ABB RAPID module: P705.mod

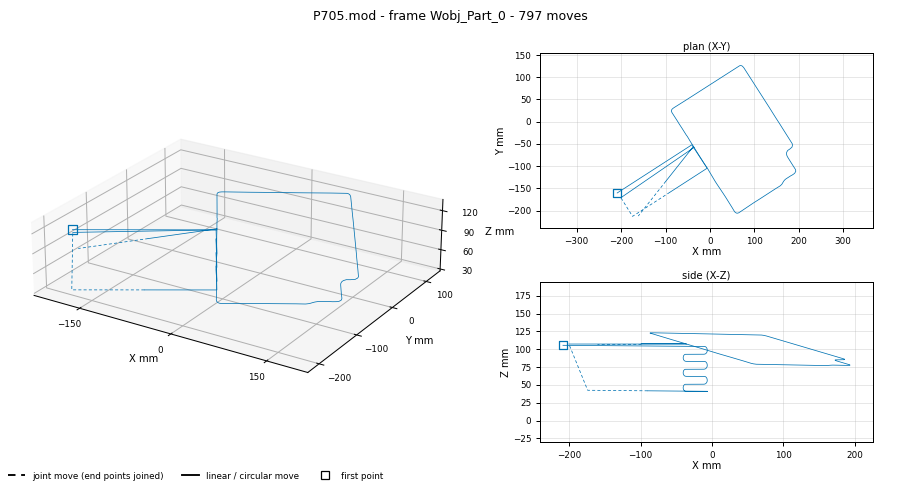
[picture p0: tool path of P705.mod in frame Wobj_Part_0, 797 of 807 moves have a stored position in this frame; points joined in program order, loops and branches not executed]
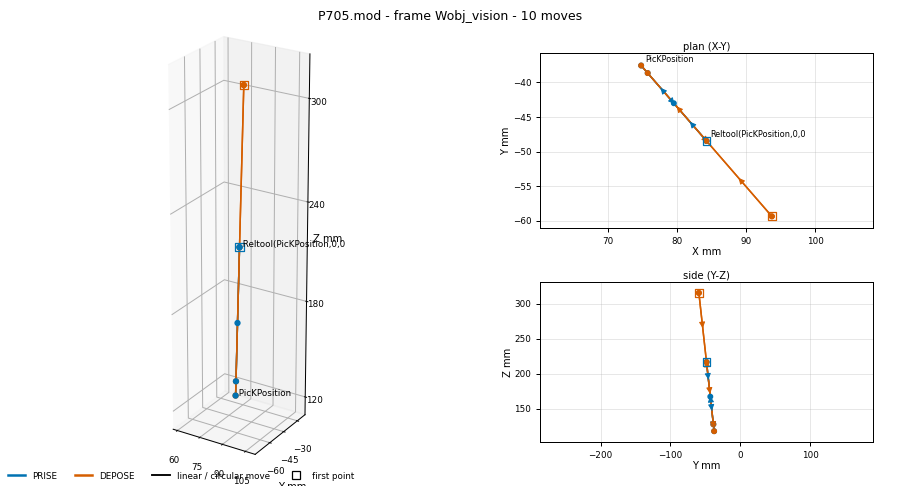
[picture p1: tool path of P705.mod in frame Wobj_vision, 10 of 807 moves have a stored position in this frame; points joined in program order, loops and branches not executed]
MODULE P705

    ! Nom         :P705
    ! Description :
    ! Créé le     :30/05/2023 11:34:18

    LOCAL CONST SPEEDDATA VitesseLente :=[10,500,0,0];
	LOCAL CONST SPEEDDATA VitesseRapide :=[30,500,0,0];
	LOCAL CONST SPEEDDATA VitesseTronconnage :=[2,500,0,0];
	LOCAL CONST SPEEDDATA VitesseTronconnageApp :=[10,500,0,0];
    !
    !Point de prise
    LOCAL PERS Robtarget PicKPosition := [[74.7644642954228,-37.5450929983313,117.878164456521],[0.0244765628567157,-0.869513599925537,0.488571722071995,0.0681518144062199],[0,0,0,0],[8.999999E+09,8.999999E+09,8.999999E+09,8.999999E+09,8.999999E+09,8.999999E+09]];
	LOCAL PERS Pose Ref := [[0,0,0],[1,0,0,0]];
    !
    !Declaration des points de meulage

    !Tr_meulage_motif_1 : Meulage d'un motif
    LOCAL CONST Robtarget Tr_meulage_motif_1_0 := [[-40.81316796875,-52.08702734375,104.0297890625],[0.61859167979337,-0.623266759536001,0.339563067143743,-0.337016028669028],[0,0,0,0],[8.999999E+09,8.999999E+09,8.999999E+09,8.999999E+09,8.999999E+09,8.999999E+09]];
    LOCAL CONST Robtarget Tr_meulage_motif_1_1 := [[-40.26262890625,-52.9218359375,104.0297890625],[0.61859167979337,-0.623266759536001,0.339563067143743,-0.337016028669028],[0,0,0,0],[8.999999E+09,8.999999E+09,8.999999E+09,8.999999E+09,8.999999E+09,8.999999E+09]];
    LOCAL CONST Robtarget Tr_meulage_motif_1_2 := [[-39.7120859375,-53.75664453125,104.0297890625],[0.61859167979337,-0.623266759536001,0.339563067143743,-0.337016028669028],[0,0,0,0],[8.999999E+09,8.999999E+09,8.999999E+09,8.999999E+09,8.999999E+09,8.999999E+09]];
    LOCAL CONST Robtarget Tr_meulage_motif_1_3 := [[-39.161546875,-54.591453125,104.0297890625],[0.61859167979337,-0.623266759536001,0.339563067143743,-0.337016028669028],[0,0,0,0],[8.999999E+09,8.999999E+09,8.999999E+09,8.999999E+09,8.999999E+09,8.999999E+09]];
    LOCAL CONST Robtarget Tr_meulage_motif_1_4 := [[-38.6110078125,-55.42626171875,104.0297890625],[0.61859167979337,-0.623266759536001,0.339563067143743,-0.337016028669028],[0,0,0,0],[8.999999E+09,8.999999E+09,8.999999E+09,8.999999E+09,8.999999E+09,8.999999E+09]];
    LOCAL CONST Robtarget Tr_meulage_motif_1_5 := [[-38.06046875,-56.2610703125,104.0297890625],[0.61859167979337,-0.623266759536001,0.339563067143743,-0.337016028669028],[0,0,0,0],[8.999999E+09,8.999999E+09,8.999999E+09,8.999999E+09,8.999999E+09,8.999999E+09]];
    LOCAL CONST Robtarget Tr_meulage_motif_1_6 := [[-37.5099296875,-57.09587890625,104.0297890625],[0.61859167979337,-0.623266759536001,0.339563067143743,-0.337016028669028],[0,0,0,0],[8.999999E+09,8.999999E+09,8.999999E+09,8.999999E+09,8.999999E+09,8.999999E+09]];
    LOCAL CONST Robtarget Tr_meulage_motif_1_7 := [[-36.95938671875,-57.9306875,104.0297890625],[0.61859167979337,-0.623266759536001,0.339563067143743,-0.337016028669028],[0,0,0,0],[8.999999E+09,8.999999E+09,8.999999E+09,8.999999E+09,8.999999E+09,8.999999E+09]];
    LOCAL CONST Robtarget Tr_meulage_motif_1_8 := [[-36.40884765625,-58.76549609375,104.0297890625],[0.61859167979337,-0.623266759536001,0.339563067143743,-0.337016028669028],[0,0,0,0],[8.999999E+09,8.999999E+09,8.999999E+09,8.999999E+09,8.999999E+09,8.999999E+09]];
    LOCAL CONST Robtarget Tr_meulage_motif_1_9 := [[-35.85830859375,-59.6003046875,104.0297890625],[0.61859167979337,-0.623266759536001,0.339563067143743,-0.337016028669028],[0,0,0,0],[8.999999E+09,8.999999E+09,8.999999E+09,8.999999E+09,8.999999E+09,8.999999E+09]];
    LOCAL CONST Robtarget Tr_meulage_motif_1_10 := [[-35.30776953125,-60.43511328125,104.0297890625],[0.61859167979337,-0.623266759536001,0.339563067143743,-0.337016028669028],[0,0,0,0],[8.999999E+09,8.999999E+09,8.999999E+09,8.999999E+09,8.999999E+09,8.999999E+09]];
    LOCAL CONST Robtarget Tr_meulage_motif_1_11 := [[-34.75723046875,-61.269921875,104.0297890625],[0.61859167979337,-0.623266759536001,0.339563067143743,-0.337016028669028],[0,0,0,0],[8.999999E+09,8.999999E+09,8.999999E+09,8.999999E+09,8.999999E+09,8.999999E+09]];
    LOCAL CONST Robtarget Tr_meulage_motif_1_12 := [[-34.2066875,-62.104734375,104.0297890625],[0.61859167979337,-0.623266759536001,0.339563067143743,-0.337016028669028],[0,0,0,0],[8.999999E+09,8.999999E+09,8.999999E+09,8.999999E+09,8.999999E+09,8.999999E+09]];
    LOCAL CONST Robtarget Tr_meulage_motif_1_13 := [[-33.6561484375,-62.93954296875,104.0297890625],[0.61859167979337,-0.623266759536001,0.339563067143743,-0.337016028669028],[0,0,0,0],[8.999999E+09,8.999999E+09,8.999999E+09,8.999999E+09,8.999999E+09,8.999999E+09]];
    LOCAL CONST Robtarget Tr_meulage_motif_1_14 := [[-33.105609375,-63.7743515625,104.0297890625],[0.61859167979337,-0.623266759536001,0.339563067143743,-0.337016028669028],[0,0,0,0],[8.999999E+09,8.999999E+09,8.999999E+09,8.999999E+09,8.999999E+09,8.999999E+09]];
    LOCAL CONST Robtarget Tr_meulage_motif_1_15 := [[-32.555068359375,-64.60916015625,104.029796875],[0.61859167979337,-0.623266759536001,0.339563067143743,-0.337016028669028],[0,0,0,0],[8.999999E+09,8.999999E+09,8.999999E+09,8.999999E+09,8.999999E+09,8.999999E+09]];
    LOCAL CONST Robtarget Tr_meulage_motif_1_16 := [[-32.004529296875,-65.44396875,104.029796875],[0.61859167979337,-0.623266759536001,0.339563067143743,-0.337016028669028],[0,0,0,0],[8.999999E+09,8.999999E+09,8.999999E+09,8.999999E+09,8.999999E+09,8.999999E+09]];
    LOCAL CONST Robtarget Tr_meulage_motif_1_17 := [[-31.453990234375,-66.2787734375,104.029796875],[0.61859167979337,-0.623266759536001,0.339563067143743,-0.337016028669028],[0,0,0,0],[8.999999E+09,8.999999E+09,8.999999E+09,8.999999E+09,8.999999E+09,8.999999E+09]];
    LOCAL CONST Robtarget Tr_meulage_motif_1_18 := [[-30.90344921875,-67.1135859375,104.029796875],[0.61859167979337,-0.623266759536001,0.339563067143743,-0.337016028669028],[0,0,0,0],[8.999999E+09,8.999999E+09,8.999999E+09,8.999999E+09,8.999999E+09,8.999999E+09]];
    LOCAL CONST Robtarget Tr_meulage_motif_1_19 := [[-30.35291015625,-67.9483984375,104.029796875],[0.61859167979337,-0.623266759536001,0.339563067143743,-0.337016028669028],[0,0,0,0],[8.999999E+09,8.999999E+09,8.999999E+09,8.999999E+09,8.999999E+09,8.999999E+09]];
    LOCAL CONST Robtarget Tr_meulage_motif_1_20 := [[-29.802369140625,-68.783203125,104.029796875],[0.61859167979337,-0.623266759536001,0.339563067143743,-0.337016028669028],[0,0,0,0],[8.999999E+09,8.999999E+09,8.999999E+09,8.999999E+09,8.999999E+09,8.999999E+09]];
    LOCAL CONST Robtarget Tr_meulage_motif_1_21 := [[-29.251830078125,-69.618015625,104.029796875],[0.61859167979337,-0.623266759536001,0.339563067143743,-0.337016028669028],[0,0,0,0],[8.999999E+09,8.999999E+09,8.999999E+09,8.999999E+09,8.999999E+09,8.999999E+09]];
    LOCAL CONST Robtarget Tr_meulage_motif_1_22 := [[-28.7012890625,-70.4528203125,104.029796875],[0.61859167979337,-0.623266759536001,0.339563067143743,-0.337016028669028],[0,0,0,0],[8.999999E+09,8.999999E+09,8.999999E+09,8.999999E+09,8.999999E+09,8.999999E+09]];
    LOCAL CONST Robtarget Tr_meulage_motif_1_23 := [[-28.15075,-71.2876328125,104.029796875],[0.61859167979337,-0.623266759536001,0.339563067143743,-0.337016028669028],[0,0,0,0],[8.999999E+09,8.999999E+09,8.999999E+09,8.999999E+09,8.999999E+09,8.999999E+09]];
    LOCAL CONST Robtarget Tr_meulage_motif_1_24 := [[-27.6002109375,-72.1224375,104.029796875],[0.61859167979337,-0.623266759536001,0.339563067143743,-0.337016028669028],[0,0,0,0],[8.999999E+09,8.999999E+09,8.999999E+09,8.999999E+09,8.999999E+09,8.999999E+09]];
    LOCAL CONST Robtarget Tr_meulage_motif_1_25 := [[-27.049669921875,-72.95725,104.029796875],[0.61859167979337,-0.623266759536001,0.339563067143743,-0.337016028669028],[0,0,0,0],[8.999999E+09,8.999999E+09,8.999999E+09,8.999999E+09,8.999999E+09,8.999999E+09]];
    LOCAL CONST Robtarget Tr_meulage_motif_1_26 := [[-26.499130859375,-73.7920546875,104.029796875],[0.61859167979337,-0.623266759536001,0.339563067143743,-0.337016028669028],[0,0,0,0],[8.999999E+09,8.999999E+09,8.999999E+09,8.999999E+09,8.999999E+09,8.999999E+09]];
    LOCAL CONST Robtarget Tr_meulage_motif_1_27 := [[-25.94858984375,-74.6268671875,104.029796875],[0.61859167979337,-0.623266759536001,0.339563067143743,-0.337016028669028],[0,0,0,0],[8.999999E+09,8.999999E+09,8.999999E+09,8.999999E+09,8.999999E+09,8.999999E+09]];
    LOCAL CONST Robtarget Tr_meulage_motif_1_28 := [[-25.39805078125,-75.461671875,104.029796875],[0.61859167979337,-0.623266759536001,0.339563067143743,-0.337016028669028],[0,0,0,0],[8.999999E+09,8.999999E+09,8.999999E+09,8.999999E+09,8.999999E+09,8.999999E+09]];
    LOCAL CONST Robtarget Tr_meulage_motif_1_29 := [[-24.84751171875,-76.296484375,104.029796875],[0.61859167979337,-0.623266759536001,0.339563067143743,-0.337016028669028],[0,0,0,0],[8.999999E+09,8.999999E+09,8.999999E+09,8.999999E+09,8.999999E+09,8.999999E+09]];
    LOCAL CONST Robtarget Tr_meulage_motif_1_30 := [[-24.296970703125,-77.1312890625,104.029796875],[0.61859167979337,-0.623266759536001,0.339563067143743,-0.337016028669028],[0,0,0,0],[8.999999E+09,8.999999E+09,8.999999E+09,8.999999E+09,8.999999E+09,8.999999E+09]];
    LOCAL CONST Robtarget Tr_meulage_motif_1_31 := [[-23.746431640625,-77.9661015625,104.029796875],[0.61859167979337,-0.623266759536001,0.339563067143743,-0.337016028669028],[0,0,0,0],[8.999999E+09,8.999999E+09,8.999999E+09,8.999999E+09,8.999999E+09,8.999999E+09]];
    LOCAL CONST Robtarget Tr_meulage_motif_1_32 := [[-23.195890625,-78.80090625,104.029796875],[0.61859167979337,-0.623266759536001,0.339563067143743,-0.337016028669028],[0,0,0,0],[8.999999E+09,8.999999E+09,8.999999E+09,8.999999E+09,8.999999E+09,8.999999E+09]];
    LOCAL CONST Robtarget Tr_meulage_motif_1_33 := [[-22.6453515625,-79.63571875,104.029796875],[0.61859167979337,-0.623266759536001,0.339563067143743,-0.337016028669028],[0,0,0,0],[8.999999E+09,8.999999E+09,8.999999E+09,8.999999E+09,8.999999E+09,8.999999E+09]];
    LOCAL CONST Robtarget Tr_meulage_motif_1_34 := [[-22.0948125,-80.47053125,104.029796875],[0.61859167979337,-0.623266759536001,0.339563067143743,-0.337016028669028],[0,0,0,0],[8.999999E+09,8.999999E+09,8.999999E+09,8.999999E+09,8.999999E+09,8.999999E+09]];
    LOCAL CONST Robtarget Tr_meulage_motif_1_35 := [[-21.544271484375,-81.3053359375,104.029796875],[0.61859167979337,-0.623266759536001,0.339563067143743,-0.337016028669028],[0,0,0,0],[8.999999E+09,8.999999E+09,8.999999E+09,8.999999E+09,8.999999E+09,8.999999E+09]];
    LOCAL CONST Robtarget Tr_meulage_motif_1_36 := [[-20.993732421875,-82.1401484375,104.029796875],[0.61859167979337,-0.623266759536001,0.339563067143743,-0.337016028669028],[0,0,0,0],[8.999999E+09,8.999999E+09,8.999999E+09,8.999999E+09,8.999999E+09,8.999999E+09]];
    LOCAL CONST Robtarget Tr_meulage_motif_1_37 := [[-20.44319140625,-82.974953125,104.029796875],[0.61859167979337,-0.623266759536001,0.339563067143743,-0.337016028669028],[0,0,0,0],[8.999999E+09,8.999999E+09,8.999999E+09,8.999999E+09,8.999999E+09,8.999999E+09]];
    LOCAL CONST Robtarget Tr_meulage_motif_1_38 := [[-19.89265234375,-83.809765625,104.029796875],[0.61859167979337,-0.623266759536001,0.339563067143743,-0.337016028669028],[0,0,0,0],[8.999999E+09,8.999999E+09,8.999999E+09,8.999999E+09,8.999999E+09,8.999999E+09]];
    LOCAL CONST Robtarget Tr_meulage_motif_1_39 := [[-19.342111328125,-84.6445703125,104.029796875],[0.61859167979337,-0.623266759536001,0.339563067143743,-0.337016028669028],[0,0,0,0],[8.999999E+09,8.999999E+09,8.999999E+09,8.999999E+09,8.999999E+09,8.999999E+09]];
    LOCAL CONST Robtarget Tr_meulage_motif_1_40 := [[-18.791572265625,-85.4793828125,104.029796875],[0.61859167979337,-0.623266759536001,0.339563067143743,-0.337016028669028],[0,0,0,0],[8.999999E+09,8.999999E+09,8.999999E+09,8.999999E+09,8.999999E+09,8.999999E+09]];
    LOCAL CONST Robtarget Tr_meulage_motif_1_41 := [[-18.241033203125,-86.3141875,104.029796875],[0.61859167979337,-0.623266759536001,0.339563067143743,-0.337016028669028],[0,0,0,0],[8.999999E+09,8.999999E+09,8.999999E+09,8.999999E+09,8.999999E+09,8.999999E+09]];
    LOCAL CONST Robtarget Tr_meulage_motif_1_42 := [[-17.6904921875,-87.149,104.029796875],[0.61859167979337,-0.623266759536001,0.339563067143743,-0.337016028669028],[0,0,0,0],[8.999999E+09,8.999999E+09,8.999999E+09,8.999999E+09,8.999999E+09,8.999999E+09]];
    LOCAL CONST Robtarget Tr_meulage_motif_1_43 := [[-17.139953125,-87.9838046875,104.029796875],[0.61859167979337,-0.623266759536001,0.339563067143743,-0.337016028669028],[0,0,0,0],[8.999999E+09,8.999999E+09,8.999999E+09,8.999999E+09,8.999999E+09,8.999999E+09]];
    LOCAL CONST Robtarget Tr_meulage_motif_1_44 := [[-16.589412109375,-88.8186171875,104.029796875],[0.61859167979337,-0.623266759536001,0.339563067143743,-0.337016028669028],[0,0,0,0],[8.999999E+09,8.999999E+09,8.999999E+09,8.999999E+09,8.999999E+09,8.999999E+09]];
    LOCAL CONST Robtarget Tr_meulage_motif_1_45 := [[-16.038873046875,-89.653421875,104.029796875],[0.61859167979337,-0.623266759536001,0.339563067143743,-0.337016028669028],[0,0,0,0],[8.999999E+09,8.999999E+09,8.999999E+09,8.999999E+09,8.999999E+09,8.999999E+09]];
    LOCAL CONST Robtarget Tr_meulage_motif_1_46 := [[-15.4883330078125,-90.488234375,104.029796875],[0.61859167979337,-0.623266759536001,0.339563067143743,-0.337016028669028],[0,0,0,0],[8.999999E+09,8.999999E+09,8.999999E+09,8.999999E+09,8.999999E+09,8.999999E+09]];
    LOCAL CONST Robtarget Tr_meulage_motif_1_47 := [[-14.93779296875,-91.323046875,104.029796875],[0.61859167979337,-0.623266759536001,0.339563067143743,-0.337016028669028],[0,0,0,0],[8.999999E+09,8.999999E+09,8.999999E+09,8.999999E+09,8.999999E+09,8.999999E+09]];
    LOCAL CONST Robtarget Tr_meulage_motif_1_48 := [[-14.38725390625,-92.1578515625,104.029796875],[0.61859167979337,-0.623266759536001,0.339563067143743,-0.337016028669028],[0,0,0,0],[8.999999E+09,8.999999E+09,8.999999E+09,8.999999E+09,8.999999E+09,8.999999E+09]];
    LOCAL CONST Robtarget Tr_meulage_motif_1_49 := [[-13.8367138671875,-92.9926640625,104.029796875],[0.61859167979337,-0.623266759536001,0.339563067143743,-0.337016028669028],[0,0,0,0],[8.999999E+09,8.999999E+09,8.999999E+09,8.999999E+09,8.999999E+09,8.999999E+09]];
    LOCAL CONST Robtarget Tr_meulage_motif_1_50 := [[-13.286173828125,-93.82746875,104.029796875],[0.61859167979337,-0.623266759536001,0.339563067143743,-0.337016028669028],[0,0,0,0],[8.999999E+09,8.999999E+09,8.999999E+09,8.999999E+09,8.999999E+09,8.999999E+09]];
    LOCAL CONST Robtarget Tr_meulage_motif_1_51 := [[-12.7356337890625,-94.66228125,104.029796875],[0.61859167979337,-0.623266759536001,0.339563067143743,-0.337016028669028],[0,0,0,0],[8.999999E+09,8.999999E+09,8.999999E+09,8.999999E+09,8.999999E+09,8.999999E+09]];
    LOCAL CONST Robtarget Tr_meulage_motif_1_52 := [[-12.18509375,-95.4970859375,104.029796875],[0.61859167979337,-0.623266759536001,0.339563067143743,-0.337016028669028],[0,0,0,0],[8.999999E+09,8.999999E+09,8.999999E+09,8.999999E+09,8.999999E+09,8.999999E+09]];
    LOCAL CONST Robtarget Tr_meulage_motif_1_53 := [[-11.6345537109375,-96.3318984375,104.029796875],[0.61859167979337,-0.623266759536001,0.339563067143743,-0.337016028669028],[0,0,0,0],[8.999999E+09,8.999999E+09,8.999999E+09,8.999999E+09,8.999999E+09,8.999999E+09]];
    LOCAL CONST Robtarget Tr_meulage_motif_1_54 := [[-11.0840146484375,-97.166703125,104.029796875],[0.61859167979337,-0.623266759536001,0.339563067143743,-0.337016028669028],[0,0,0,0],[8.999999E+09,8.999999E+09,8.999999E+09,8.999999E+09,8.999999E+09,8.999999E+09]];
    LOCAL CONST Robtarget Tr_meulage_motif_1_55 := [[-10.533474609375,-98.001515625,104.029796875],[0.61859167979337,-0.623266759536001,0.339563067143743,-0.337016028669028],[0,0,0,0],[8.999999E+09,8.999999E+09,8.999999E+09,8.999999E+09,8.999999E+09,8.999999E+09]];
    LOCAL CONST Robtarget Tr_meulage_motif_1_56 := [[-9.987146484375,-98.8301875,103.919203125],[0.61859167979337,-0.623266759536001,0.339563067143743,-0.337016028669028],[0,0,0,0],[8.999999E+09,8.999999E+09,8.999999E+09,8.999999E+09,8.999999E+09,8.999999E+09]];
    LOCAL CONST Robtarget Tr_meulage_motif_1_57 := [[-9.4662841796875,-99.620484375,103.708015625],[0.61859167979337,-0.623266759536001,0.339563067143743,-0.337016028669028],[0,0,0,0],[8.999999E+09,8.999999E+09,8.999999E+09,8.999999E+09,8.999999E+09,8.999999E+09]];
    LOCAL CONST Robtarget Tr_meulage_motif_1_58 := [[-8.9971162109375,-100.33253125,103.436171875],[0.61859167979337,-0.623266759536001,0.339563067143743,-0.337016028669028],[0,0,0,0],[8.999999E+09,8.999999E+09,8.999999E+09,8.999999E+09,8.999999E+09,8.999999E+09]];
    LOCAL CONST Robtarget Tr_meulage_motif_1_59 := [[-8.5845380859375,-100.95878125,103.160234375],[0.61859167979337,-0.623266759536001,0.339563067143743,-0.337016028669028],[0,0,0,0],[8.999999E+09,8.999999E+09,8.999999E+09,8.999999E+09,8.999999E+09,8.999999E+09]];
    LOCAL CONST Robtarget Tr_meulage_motif_1_60 := [[-7.97901220703125,-101.878390625,102.544109375],[0.61859167979337,-0.623266759536001,0.339563067143743,-0.337016028669028],[0,0,0,0],[8.999999E+09,8.999999E+09,8.999999E+09,8.999999E+09,8.999999E+09,8.999999E+09]];
    LOCAL CONST Robtarget Tr_meulage_motif_1_61 := [[-7.41622607421875,-102.73371875,101.696453125],[0.61859167979337,-0.623266759536001,0.339563067143743,-0.337016028669028],[0,0,0,0],[8.999999E+09,8.999999E+09,8.999999E+09,8.999999E+09,8.999999E+09,8.999999E+09]];
    LOCAL CONST Robtarget Tr_meulage_motif_1_62 := [[-6.95064208984375,-103.4420625,100.6725859375],[0.61859167979337,-0.623266759536001,0.339563067143743,-0.337016028669028],[0,0,0,0],[8.999999E+09,8.999999E+09,8.999999E+09,8.999999E+09,8.999999E+09,8.999999E+09]];
    LOCAL CONST Robtarget Tr_meulage_motif_1_63 := [[-6.68307470703125,-103.850359375,99.5563984375],[0.61859167979337,-0.623266759536001,0.339563067143743,-0.337016028669028],[0,0,0,0],[8.999999E+09,8.999999E+09,8.999999E+09,8.999999E+09,8.999999E+09,8.999999E+09]];
    LOCAL CONST Robtarget Tr_meulage_motif_1_64 := [[-6.6689130859375,-103.8734375,98.8604296875],[0.61859167979337,-0.623266759536001,0.339563067143743,-0.337016028669028],[0,0,0,0],[8.999999E+09,8.999999E+09,8.999999E+09,8.999999E+09,8.999999E+09,8.999999E+09]];
    LOCAL CONST Robtarget Tr_meulage_motif_1_65 := [[-6.66961376953125,-103.87390625,98.1991796875],[0.61859167979337,-0.623266759536001,0.339563067143743,-0.337016028669028],[0,0,0,0],[8.999999E+09,8.999999E+09,8.999999E+09,8.999999E+09,8.999999E+09,8.999999E+09]];
    LOCAL CONST Robtarget Tr_meulage_motif_1_66 := [[-6.70052490234375,-103.8285546875,97.5380859375],[0.61859167979337,-0.623266759536001,0.339563067143743,-0.337016028669028],[0,0,0,0],[8.999999E+09,8.999999E+09,8.999999E+09,8.999999E+09,8.999999E+09,8.999999E+09]];
    LOCAL CONST Robtarget Tr_meulage_motif_1_67 := [[-6.97598095703125,-103.41340625,96.4363359375],[0.61859167979337,-0.623266759536001,0.339563067143743,-0.337016028669028],[0,0,0,0],[8.999999E+09,8.999999E+09,8.999999E+09,8.999999E+09,8.999999E+09,8.999999E+09]];
    LOCAL CONST Robtarget Tr_meulage_motif_1_68 := [[-7.44865380859375,-102.6989921875,95.4297109375],[0.61859167979337,-0.623266759536001,0.339563067143743,-0.337016028669028],[0,0,0,0],[8.999999E+09,8.999999E+09,8.999999E+09,8.999999E+09,8.999999E+09,8.999999E+09]];
    LOCAL CONST Robtarget Tr_meulage_motif_1_69 := [[-8.012974609375,-101.8451953125,94.6008359375],[0.61859167979337,-0.623266759536001,0.339563067143743,-0.337016028669028],[0,0,0,0],[8.999999E+09,8.999999E+09,8.999999E+09,8.999999E+09,8.999999E+09,8.999999E+09]];
    LOCAL CONST Robtarget Tr_meulage_motif_1_70 := [[-8.3916494140625,-101.27190625,94.2050859375],[0.61859167979337,-0.623266759536001,0.339563067143743,-0.337016028669028],[0,0,0,0],[8.999999E+09,8.999999E+09,8.999999E+09,8.999999E+09,8.999999E+09,8.999999E+09]];
    LOCAL CONST Robtarget Tr_meulage_motif_1_71 := [[-9.02977734375,-100.30540625,93.7175546875],[0.61859167979337,-0.623266759536001,0.339563067143743,-0.337016028669028],[0,0,0,0],[8.999999E+09,8.999999E+09,8.999999E+09,8.999999E+09,8.999999E+09,8.999999E+09]];
    LOCAL CONST Robtarget Tr_meulage_motif_1_72 := [[-9.4952802734375,-99.60015625,93.4534609375],[0.61859167979337,-0.623266759536001,0.339563067143743,-0.337016028669028],[0,0,0,0],[8.999999E+09,8.999999E+09,8.999999E+09,8.999999E+09,8.999999E+09,8.999999E+09]];
    LOCAL CONST Robtarget Tr_meulage_motif_1_73 := [[-10.008599609375,-98.8222578125,93.2489921875],[0.61859167979337,-0.623266759536001,0.339563067143743,-0.337016028669028],[0,0,0,0],[8.999999E+09,8.999999E+09,8.999999E+09,8.999999E+09,8.999999E+09,8.999999E+09]];
    LOCAL CONST Robtarget Tr_meulage_motif_1_74 := [[-10.5491044921875,-98.0029140625,93.1403984375],[0.61859167979337,-0.623266759536001,0.339563067143743,-0.337016028669028],[0,0,0,0],[8.999999E+09,8.999999E+09,8.999999E+09,8.999999E+09,8.999999E+09,8.999999E+09]];
    LOCAL CONST Robtarget Tr_meulage_motif_1_75 := [[-11.0956669921875,-97.174390625,93.0298046875],[0.61859167979337,-0.623266759536001,0.339563067143743,-0.337016028669028],[0,0,0,0],[8.999999E+09,8.999999E+09,8.999999E+09,8.999999E+09,8.999999E+09,8.999999E+09]];
    LOCAL CONST Robtarget Tr_meulage_motif_1_76 := [[-11.6462060546875,-96.3395859375,93.0298046875],[0.61859167979337,-0.623266759536001,0.339563067143743,-0.337016028669028],[0,0,0,0],[8.999999E+09,8.999999E+09,8.999999E+09,8.999999E+09,8.999999E+09,8.999999E+09]];
    LOCAL CONST Robtarget Tr_meulage_motif_1_77 := [[-12.19674609375,-95.5047734375,93.0298046875],[0.61859167979337,-0.623266759536001,0.339563067143743,-0.337016028669028],[0,0,0,0],[8.999999E+09,8.999999E+09,8.999999E+09,8.999999E+09,8.999999E+09,8.999999E+09]];
    LOCAL CONST Robtarget Tr_meulage_motif_1_78 := [[-12.7472861328125,-94.6699609375,93.0298046875],[0.61859167979337,-0.623266759536001,0.339563067143743,-0.337016028669028],[0,0,0,0],[8.999999E+09,8.999999E+09,8.999999E+09,8.999999E+09,8.999999E+09,8.999999E+09]];
    LOCAL CONST Robtarget Tr_meulage_motif_1_79 := [[-13.297826171875,-93.83515625,93.0298046875],[0.61859167979337,-0.623266759536001,0.339563067143743,-0.337016028669028],[0,0,0,0],[8.999999E+09,8.999999E+09,8.999999E+09,8.999999E+09,8.999999E+09,8.999999E+09]];
    LOCAL CONST Robtarget Tr_meulage_motif_1_80 := [[-13.8483662109375,-93.00034375,93.0298046875],[0.61859167979337,-0.623266759536001,0.339563067143743,-0.337016028669028],[0,0,0,0],[8.999999E+09,8.999999E+09,8.999999E+09,8.999999E+09,8.999999E+09,8.999999E+09]];
    LOCAL CONST Robtarget Tr_meulage_motif_1_81 := [[-14.39890625,-92.1655390625,93.0298046875],[0.61859167979337,-0.623266759536001,0.339563067143743,-0.337016028669028],[0,0,0,0],[8.999999E+09,8.999999E+09,8.999999E+09,8.999999E+09,8.999999E+09,8.999999E+09]];
    LOCAL CONST Robtarget Tr_meulage_motif_1_82 := [[-14.9494453125,-91.3307265625,93.0298046875],[0.61859167979337,-0.623266759536001,0.339563067143743,-0.337016028669028],[0,0,0,0],[8.999999E+09,8.999999E+09,8.999999E+09,8.999999E+09,8.999999E+09,8.999999E+09]];
    LOCAL CONST Robtarget Tr_meulage_motif_1_83 := [[-15.4999853515625,-90.495921875,93.0298046875],[0.61859167979337,-0.623266759536001,0.339563067143743,-0.337016028669028],[0,0,0,0],[8.999999E+09,8.999999E+09,8.999999E+09,8.999999E+09,8.999999E+09,8.999999E+09]];
    LOCAL CONST Robtarget Tr_meulage_motif_1_84 := [[-16.050525390625,-89.661109375,93.0298046875],[0.61859167979337,-0.623266759536001,0.339563067143743,-0.337016028669028],[0,0,0,0],[8.999999E+09,8.999999E+09,8.999999E+09,8.999999E+09,8.999999E+09,8.999999E+09]];
    LOCAL CONST Robtarget Tr_meulage_motif_1_85 := [[-16.601064453125,-88.8263046875,93.0298046875],[0.61859167979337,-0.623266759536001,0.339563067143743,-0.337016028669028],[0,0,0,0],[8.999999E+09,8.999999E+09,8.999999E+09,8.999999E+09,8.999999E+09,8.999999E+09]];
    LOCAL CONST Robtarget Tr_meulage_motif_1_86 := [[-17.15160546875,-87.9914921875,93.0298046875],[0.61859167979337,-0.623266759536001,0.339563067143743,-0.337016028669028],[0,0,0,0],[8.999999E+09,8.999999E+09,8.999999E+09,8.999999E+09,8.999999E+09,8.999999E+09]];
    LOCAL CONST Robtarget Tr_meulage_motif_1_87 := [[-17.70214453125,-87.1566875,93.0298046875],[0.61859167979337,-0.623266759536001,0.339563067143743,-0.337016028669028],[0,0,0,0],[8.999999E+09,8.999999E+09,8.999999E+09,8.999999E+09,8.999999E+09,8.999999E+09]];
    LOCAL CONST Robtarget Tr_meulage_motif_1_88 := [[-18.252685546875,-86.321875,93.0298046875],[0.61859167979337,-0.623266759536001,0.339563067143743,-0.337016028669028],[0,0,0,0],[8.999999E+09,8.999999E+09,8.999999E+09,8.999999E+09,8.999999E+09,8.999999E+09]];
    LOCAL CONST Robtarget Tr_meulage_motif_1_89 := [[-18.803224609375,-85.4870703125,93.0298046875],[0.61859167979337,-0.623266759536001,0.339563067143743,-0.337016028669028],[0,0,0,0],[8.999999E+09,8.999999E+09,8.999999E+09,8.999999E+09,8.999999E+09,8.999999E+09]];
    LOCAL CONST Robtarget Tr_meulage_motif_1_90 := [[-19.353763671875,-84.6522578125,93.0298046875],[0.61859167979337,-0.623266759536001,0.339563067143743,-0.337016028669028],[0,0,0,0],[8.999999E+09,8.999999E+09,8.999999E+09,8.999999E+09,8.999999E+09,8.999999E+09]];
    LOCAL CONST Robtarget Tr_meulage_motif_1_91 := [[-19.9043046875,-83.817453125,93.0298046875],[0.61859167979337,-0.623266759536001,0.339563067143743,-0.337016028669028],[0,0,0,0],[8.999999E+09,8.999999E+09,8.999999E+09,8.999999E+09,8.999999E+09,8.999999E+09]];
    LOCAL CONST Robtarget Tr_meulage_motif_1_92 := [[-20.45484375,-82.982640625,93.0298046875],[0.61859167979337,-0.623266759536001,0.339563067143743,-0.337016028669028],[0,0,0,0],[8.999999E+09,8.999999E+09,8.999999E+09,8.999999E+09,8.999999E+09,8.999999E+09]];
    LOCAL CONST Robtarget Tr_meulage_motif_1_93 := [[-21.005384765625,-82.147828125,93.0298046875],[0.61859167979337,-0.623266759536001,0.339563067143743,-0.337016028669028],[0,0,0,0],[8.999999E+09,8.999999E+09,8.999999E+09,8.999999E+09,8.999999E+09,8.999999E+09]];
    LOCAL CONST Robtarget Tr_meulage_motif_1_94 := [[-21.555923828125,-81.3130234375,93.0298046875],[0.61859167979337,-0.623266759536001,0.339563067143743,-0.337016028669028],[0,0,0,0],[8.999999E+09,8.999999E+09,8.999999E+09,8.999999E+09,8.999999E+09,8.999999E+09]];
    LOCAL CONST Robtarget Tr_meulage_motif_1_95 := [[-22.10646484375,-80.4782109375,93.0298046875],[0.61859167979337,-0.623266759536001,0.339563067143743,-0.337016028669028],[0,0,0,0],[8.999999E+09,8.999999E+09,8.999999E+09,8.999999E+09,8.999999E+09,8.999999E+09]];
    LOCAL CONST Robtarget Tr_meulage_motif_1_96 := [[-22.65700390625,-79.64340625,93.0298046875],[0.61859167979337,-0.623266759536001,0.339563067143743,-0.337016028669028],[0,0,0,0],[8.999999E+09,8.999999E+09,8.999999E+09,8.999999E+09,8.999999E+09,8.999999E+09]];
    LOCAL CONST Robtarget Tr_meulage_motif_1_97 := [[-23.20754296875,-78.80859375,93.0298046875],[0.61859167979337,-0.623266759536001,0.339563067143743,-0.337016028669028],[0,0,0,0],[8.999999E+09,8.999999E+09,8.999999E+09,8.999999E+09,8.999999E+09,8.999999E+09]];
    LOCAL CONST Robtarget Tr_meulage_motif_1_98 := [[-23.758083984375,-77.9737890625,93.0298046875],[0.61859167979337,-0.623266759536001,0.339563067143743,-0.337016028669028],[0,0,0,0],[8.999999E+09,8.999999E+09,8.999999E+09,8.999999E+09,8.999999E+09,8.999999E+09]];
    LOCAL CONST Robtarget Tr_meulage_motif_1_99 := [[-24.308623046875,-77.1389765625,93.0298046875],[0.61859167979337,-0.623266759536001,0.339563067143743,-0.337016028669028],[0,0,0,0],[8.999999E+09,8.999999E+09,8.999999E+09,8.999999E+09,8.999999E+09,8.999999E+09]];
    LOCAL CONST Robtarget Tr_meulage_motif_1_100 := [[-24.8591640625,-76.304171875,93.0298046875],[0.61859167979337,-0.623266759536001,0.339563067143743,-0.337016028669028],[0,0,0,0],[8.999999E+09,8.999999E+09,8.999999E+09,8.999999E+09,8.999999E+09,8.999999E+09]];
    LOCAL CONST Robtarget Tr_meulage_motif_1_101 := [[-25.409703125,-75.469359375,93.0298046875],[0.61859167979337,-0.623266759536001,0.339563067143743,-0.337016028669028],[0,0,0,0],[8.999999E+09,8.999999E+09,8.999999E+09,8.999999E+09,8.999999E+09,8.999999E+09]];
    LOCAL CONST Robtarget Tr_meulage_motif_1_102 := [[-25.9602421875,-74.6345546875,93.0298046875],[0.61859167979337,-0.623266759536001,0.339563067143743,-0.337016028669028],[0,0,0,0],[8.999999E+09,8.999999E+09,8.999999E+09,8.999999E+09,8.999999E+09,8.999999E+09]];
    LOCAL CONST Robtarget Tr_meulage_motif_1_103 := [[-26.510783203125,-73.7997421875,93.0298046875],[0.61859167979337,-0.623266759536001,0.339563067143743,-0.337016028669028],[0,0,0,0],[8.999999E+09,8.999999E+09,8.999999E+09,8.999999E+09,8.999999E+09,8.999999E+09]];
    LOCAL CONST Robtarget Tr_meulage_motif_1_104 := [[-27.061322265625,-72.9649375,93.0298046875],[0.61859167979337,-0.623266759536001,0.339563067143743,-0.337016028669028],[0,0,0,0],[8.999999E+09,8.999999E+09,8.999999E+09,8.999999E+09,8.999999E+09,8.999999E+09]];
    LOCAL CONST Robtarget Tr_meulage_motif_1_105 := [[-27.61186328125,-72.130125,93.0298046875],[0.61859167979337,-0.623266759536001,0.339563067143743,-0.337016028669028],[0,0,0,0],[8.999999E+09,8.999999E+09,8.999999E+09,8.999999E+09,8.999999E+09,8.999999E+09]];
    LOCAL CONST Robtarget Tr_meulage_motif_1_106 := [[-28.16240234375,-71.2953125,93.0298046875],[0.61859167979337,-0.623266759536001,0.339563067143743,-0.337016028669028],[0,0,0,0],[8.999999E+09,8.999999E+09,8.999999E+09,8.999999E+09,8.999999E+09,8.999999E+09]];
    LOCAL CONST Robtarget Tr_meulage_motif_1_107 := [[-28.71294140625,-70.4605078125,93.0298046875],[0.61859167979337,-0.623266759536001,0.339563067143743,-0.337016028669028],[0,0,0,0],[8.999999E+09,8.999999E+09,8.999999E+09,8.999999E+09,8.999999E+09,8.999999E+09]];
    LOCAL CONST Robtarget Tr_meulage_motif_1_108 := [[-29.263482421875,-69.6256953125,93.0298046875],[0.61859167979337,-0.623266759536001,0.339563067143743,-0.337016028669028],[0,0,0,0],[8.999999E+09,8.999999E+09,8.999999E+09,8.999999E+09,8.999999E+09,8.999999E+09]];
    LOCAL CONST Robtarget Tr_meulage_motif_1_109 := [[-29.814021484375,-68.790890625,93.0298046875],[0.61859167979337,-0.623266759536001,0.339563067143743,-0.337016028669028],[0,0,0,0],[8.999999E+09,8.999999E+09,8.999999E+09,8.999999E+09,8.999999E+09,8.999999E+09]];
    LOCAL CONST Robtarget Tr_meulage_motif_1_110 := [[-30.3645625,-67.956078125,93.0298046875],[0.61859167979337,-0.623266759536001,0.339563067143743,-0.337016028669028],[0,0,0,0],[8.999999E+09,8.999999E+09,8.999999E+09,8.999999E+09,8.999999E+09,8.999999E+09]];
    LOCAL CONST Robtarget Tr_meulage_motif_1_111 := [[-30.9151015625,-67.1212734375,93.0298046875],[0.61859167979337,-0.623266759536001,0.339563067143743,-0.337016028669028],[0,0,0,0],[8.999999E+09,8.999999E+09,8.999999E+09,8.999999E+09,8.999999E+09,8.999999E+09]];
    LOCAL CONST Robtarget Tr_meulage_motif_1_112 := [[-31.465642578125,-66.2864609375,93.0298046875],[0.61859167979337,-0.623266759536001,0.339563067143743,-0.337016028669028],[0,0,0,0],[8.999999E+09,8.999999E+09,8.999999E+09,8.999999E+09,8.999999E+09,8.999999E+09]];
    LOCAL CONST Robtarget Tr_meulage_motif_1_113 := [[-32.016181640625,-65.45165234375,93.0298046875],[0.61859167979337,-0.623266759536001,0.339563067143743,-0.337016028669028],[0,0,0,0],[8.999999E+09,8.999999E+09,8.999999E+09,8.999999E+09,8.999999E+09,8.999999E+09]];
    LOCAL CONST Robtarget Tr_meulage_motif_1_114 := [[-32.566720703125,-64.61684375,93.0298046875],[0.61859167979337,-0.623266759536001,0.339563067143743,-0.337016028669028],[0,0,0,0],[8.999999E+09,8.999999E+09,8.999999E+09,8.999999E+09,8.999999E+09,8.999999E+09]];
    LOCAL CONST Robtarget Tr_meulage_motif_1_115 := [[-33.11726171875,-63.78203515625,93.0298046875],[0.61859167979337,-0.623266759536001,0.339563067143743,-0.337016028669028],[0,0,0,0],[8.999999E+09,8.999999E+09,8.999999E+09,8.999999E+09,8.999999E+09,8.999999E+09]];
    LOCAL CONST Robtarget Tr_meulage_motif_1_116 := [[-33.66780078125,-62.9472265625,93.0298046875],[0.61859167979337,-0.623266759536001,0.339563067143743,-0.337016028669028],[0,0,0,0],[8.999999E+09,8.999999E+09,8.999999E+09,8.999999E+09,8.999999E+09,8.999999E+09]];
    LOCAL CONST Robtarget Tr_meulage_motif_1_117 := [[-34.21833984375,-62.11241796875,93.0298046875],[0.61859167979337,-0.623266759536001,0.339563067143743,-0.337016028669028],[0,0,0,0],[8.999999E+09,8.999999E+09,8.999999E+09,8.999999E+09,8.999999E+09,8.999999E+09]];
    LOCAL CONST Robtarget Tr_meulage_motif_1_118 := [[-34.7688828125,-61.277609375,93.0298046875],[0.61859167979337,-0.623266759536001,0.339563067143743,-0.337016028669028],[0,0,0,0],[8.999999E+09,8.999999E+09,8.999999E+09,8.999999E+09,8.999999E+09,8.999999E+09]];
    LOCAL CONST Robtarget Tr_meulage_motif_1_119 := [[-35.319421875,-60.44280078125,93.0298046875],[0.61859167979337,-0.623266759536001,0.339563067143743,-0.337016028669028],[0,0,0,0],[8.999999E+09,8.999999E+09,8.999999E+09,8.999999E+09,8.999999E+09,8.999999E+09]];
    LOCAL CONST Robtarget Tr_meulage_motif_1_120 := [[-35.8699609375,-59.6079921875,93.0298046875],[0.61859167979337,-0.623266759536001,0.339563067143743,-0.337016028669028],[0,0,0,0],[8.999999E+09,8.999999E+09,8.999999E+09,8.999999E+09,8.999999E+09,8.999999E+09]];
    LOCAL CONST Robtarget Tr_meulage_motif_1_121 := [[-36.4205,-58.77318359375,93.0298046875],[0.61859167979337,-0.623266759536001,0.339563067143743,-0.337016028669028],[0,0,0,0],[8.999999E+09,8.999999E+09,8.999999E+09,8.999999E+09,8.999999E+09,8.999999E+09]];
    LOCAL CONST Robtarget Tr_meulage_motif_1_122 := [[-36.9710390625,-57.938375,93.0298046875],[0.61859167979337,-0.623266759536001,0.339563067143743,-0.337016028669028],[0,0,0,0],[8.999999E+09,8.999999E+09,8.999999E+09,8.999999E+09,8.999999E+09,8.999999E+09]];
    LOCAL CONST Robtarget Tr_meulage_motif_1_123 := [[-37.5176015625,-57.1098515625,92.9192109375],[0.61859167979337,-0.623266759536001,0.339563067143743,-0.337016028669028],[0,0,0,0],[8.999999E+09,8.999999E+09,8.999999E+09,8.999999E+09,8.999999E+09,8.999999E+09]];
    LOCAL CONST Robtarget Tr_meulage_motif_1_124 := [[-38.0389140625,-56.3198515625,92.7080234375],[0.61859167979337,-0.623266759536001,0.339563067143743,-0.337016028669028],[0,0,0,0],[8.999999E+09,8.999999E+09,8.999999E+09,8.999999E+09,8.999999E+09,8.999999E+09]];
    LOCAL CONST Robtarget Tr_meulage_motif_1_125 := [[-38.50865625,-55.60818359375,92.4361796875],[0.61859167979337,-0.623266759536001,0.339563067143743,-0.337016028669028],[0,0,0,0],[8.999999E+09,8.999999E+09,8.999999E+09,8.999999E+09,8.999999E+09,8.999999E+09]];
    LOCAL CONST Robtarget Tr_meulage_motif_1_126 := [[-38.9006875,-55.0144296875,92.1320234375],[0.61859167979337,-0.623266759536001,0.339563067143743,-0.337016028669028],[0,0,0,0],[8.999999E+09,8.999999E+09,8.999999E+09,8.999999E+09,8.999999E+09,8.999999E+09]];
    LOCAL CONST Robtarget Tr_meulage_motif_1_127 := [[-39.47090625,-54.15130859375,91.4694921875],[0.61859167979337,-0.623266759536001,0.339563067143743,-0.337016028669028],[0,0,0,0],[8.999999E+09,8.999999E+09,8.999999E+09,8.999999E+09,8.999999E+09,8.999999E+09]];
    LOCAL CONST Robtarget Tr_meulage_motif_1_128 := [[-39.9684140625,-53.39899609375,90.5675546875],[0.61859167979337,-0.623266759536001,0.339563067143743,-0.337016028669028],[0,0,0,0],[8.999999E+09,8.999999E+09,8.999999E+09,8.999999E+09,8.999999E+09,8.999999E+09]];
    LOCAL CONST Robtarget Tr_meulage_motif_1_129 := [[-40.26404296875,-52.95312890625,89.5215234375],[0.61859167979337,-0.623266759536001,0.339563067143743,-0.337016028669028],[0,0,0,0],[8.999999E+09,8.999999E+09,8.999999E+09,8.999999E+09,8.999999E+09,8.999999E+09]];
    LOCAL CONST Robtarget Tr_meulage_motif_1_130 := [[-40.3665078125,-52.79935546875,88.8283046875],[0.61859167979337,-0.623266759536001,0.339563067143743,-0.337016028669028],[0,0,0,0],[8.999999E+09,8.999999E+09,8.999999E+09,8.999999E+09,8.999999E+09,8.999999E+09]];
    LOCAL CONST Robtarget Tr_meulage_motif_1_131 := [[-40.40247265625,-52.74659765625,88.0583046875],[0.61859167979337,-0.623266759536001,0.339563067143743,-0.337016028669028],[0,0,0,0],[8.999999E+09,8.999999E+09,8.999999E+09,8.999999E+09,8.999999E+09,8.999999E+09]];
    LOCAL CONST Robtarget Tr_meulage_motif_1_132 := [[-40.36643359375,-52.803015625,87.2884296875],[0.61859167979337,-0.623266759536001,0.339563067143743,-0.337016028669028],[0,0,0,0],[8.999999E+09,8.999999E+09,8.999999E+09,8.999999E+09,8.999999E+09,8.999999E+09]];
    LOCAL CONST Robtarget Tr_meulage_motif_1_133 := [[-40.13660546875,-53.1540703125,86.1801796875],[0.61859167979337,-0.623266759536001,0.339563067143743,-0.337016028669028],[0,0,0,0],[8.999999E+09,8.999999E+09,8.999999E+09,8.999999E+09,8.999999E+09,8.999999E+09]];
    LOCAL CONST Robtarget Tr_meulage_motif_1_134 := [[-39.90912890625,-53.5003515625,85.5944921875],[0.61859167979337,-0.623266759536001,0.339563067143743,-0.337016028669028],[0,0,0,0],[8.999999E+09,8.999999E+09,8.999999E+09,8.999999E+09,8.999999E+09,8.999999E+09]];
    LOCAL CONST Robtarget Tr_meulage_motif_1_135 := [[-39.421671875,-54.24155078125,84.7073671875],[0.61859167979337,-0.623266759536001,0.339563067143743,-0.337016028669028],[0,0,0,0],[8.999999E+09,8.999999E+09,8.999999E+09,8.999999E+09,8.999999E+09,8.999999E+09]];
    LOCAL CONST Robtarget Tr_meulage_motif_1_136 := [[-39.09966796875,-54.73077734375,84.2930546875],[0.61859167979337,-0.623266759536001,0.339563067143743,-0.337016028669028],[0,0,0,0],[8.999999E+09,8.999999E+09,8.999999E+09,8.999999E+09,8.999999E+09,8.999999E+09]];
    LOCAL CONST Robtarget Tr_meulage_motif_1_137 := [[-38.48479296875,-55.66439453125,83.7489609375],[0.61859167979337,-0.623266759536001,0.339563067143743,-0.337016028669028],[0,0,0,0],[8.999999E+09,8.999999E+09,8.999999E+09,8.999999E+09,8.999999E+09,8.999999E+09]];
    LOCAL CONST Robtarget Tr_meulage_motif_1_138 := [[-38.03058203125,-56.35381640625,83.4534609375],[0.61859167979337,-0.623266759536001,0.339563067143743,-0.337016028669028],[0,0,0,0],[8.999999E+09,8.999999E+09,8.999999E+09,8.999999E+09,8.999999E+09,8.999999E+09]];
    LOCAL CONST Robtarget Tr_meulage_motif_1_139 := [[-37.5176953125,-57.132,83.249],[0.61859167979337,-0.623266759536001,0.339563067143743,-0.337016028669028],[0,0,0,0],[8.999999E+09,8.999999E+09,8.999999E+09,8.999999E+09,8.999999E+09,8.999999E+09]];
    LOCAL CONST Robtarget Tr_meulage_motif_1_140 := [[-36.977421875,-57.9514921875,83.14040625],[0.61859167979337,-0.623266759536001,0.339563067143743,-0.337016028669028],[0,0,0,0],[8.999999E+09,8.999999E+09,8.999999E+09,8.999999E+09,8.999999E+09,8.999999E+09]];
    LOCAL CONST Robtarget Tr_meulage_motif_1_141 := [[-36.43109375,-58.780171875,83.0298125],[0.61859167979337,-0.623266759536001,0.339563067143743,-0.337016028669028],[0,0,0,0],[8.999999E+09,8.999999E+09,8.999999E+09,8.999999E+09,8.999999E+09,8.999999E+09]];
    LOCAL CONST Robtarget Tr_meulage_motif_1_142 := [[-35.8805546875,-59.61498046875,83.0298125],[0.61859167979337,-0.623266759536001,0.339563067143743,-0.337016028669028],[0,0,0,0],[8.999999E+09,8.999999E+09,8.999999E+09,8.999999E+09,8.999999E+09,8.999999E+09]];
    LOCAL CONST Robtarget Tr_meulage_motif_1_143 := [[-35.330015625,-60.4497890625,83.0298125],[0.61859167979337,-0.623266759536001,0.339563067143743,-0.337016028669028],[0,0,0,0],[8.999999E+09,8.999999E+09,8.999999E+09,8.999999E+09,8.999999E+09,8.999999E+09]];
    LOCAL CONST Robtarget Tr_meulage_motif_1_144 := [[-34.77947265625,-61.28459765625,83.0298125],[0.61859167979337,-0.623266759536001,0.339563067143743,-0.337016028669028],[0,0,0,0],[8.999999E+09,8.999999E+09,8.999999E+09,8.999999E+09,8.999999E+09,8.999999E+09]];
    LOCAL CONST Robtarget Tr_meulage_motif_1_145 := [[-34.22893359375,-62.11940625,83.0298125],[0.61859167979337,-0.623266759536001,0.339563067143743,-0.337016028669028],[0,0,0,0],[8.999999E+09,8.999999E+09,8.999999E+09,8.999999E+09,8.999999E+09,8.999999E+09]];
    LOCAL CONST Robtarget Tr_meulage_motif_1_146 := [[-33.67839453125,-62.95421484375,83.0298125],[0.61859167979337,-0.623266759536001,0.339563067143743,-0.337016028669028],[0,0,0,0],[8.999999E+09,8.999999E+09,8.999999E+09,8.999999E+09,8.999999E+09,8.999999E+09]];
    LOCAL CONST Robtarget Tr_meulage_motif_1_147 := [[-33.12785546875,-63.7890234375,83.0298125],[0.61859167979337,-0.623266759536001,0.339563067143743,-0.337016028669028],[0,0,0,0],[8.999999E+09,8.999999E+09,8.999999E+09,8.999999E+09,8.999999E+09,8.999999E+09]];
    LOCAL CONST Robtarget Tr_meulage_motif_1_148 := [[-32.577314453125,-64.62383203125,83.0298125],[0.61859167979337,-0.623266759536001,0.339563067143743,-0.337016028669028],[0,0,0,0],[8.999999E+09,8.999999E+09,8.999999E+09,8.999999E+09,8.999999E+09,8.999999E+09]];
    LOCAL CONST Robtarget Tr_meulage_motif_1_149 := [[-32.026775390625,-65.458640625,83.0298125],[0.61859167979337,-0.623266759536001,0.339563067143743,-0.337016028669028],[0,0,0,0],[8.999999E+09,8.999999E+09,8.999999E+09,8.999999E+09,8.999999E+09,8.999999E+09]];
    LOCAL CONST Robtarget Tr_meulage_motif_1_150 := [[-31.476234375,-66.293453125,83.0298125],[0.61859167979337,-0.623266759536001,0.339563067143743,-0.337016028669028],[0,0,0,0],[8.999999E+09,8.999999E+09,8.999999E+09,8.999999E+09,8.999999E+09,8.999999E+09]];
    LOCAL CONST Robtarget Tr_meulage_motif_1_151 := [[-30.9256953125,-67.1282578125,83.0298125],[0.61859167979337,-0.623266759536001,0.339563067143743,-0.337016028669028],[0,0,0,0],[8.999999E+09,8.999999E+09,8.999999E+09,8.999999E+09,8.999999E+09,8.999999E+09]];
    LOCAL CONST Robtarget Tr_meulage_motif_1_152 := [[-30.375154296875,-67.9630703125,83.0298125],[0.61859167979337,-0.623266759536001,0.339563067143743,-0.337016028669028],[0,0,0,0],[8.999999E+09,8.999999E+09,8.999999E+09,8.999999E+09,8.999999E+09,8.999999E+09]];
    LOCAL CONST Robtarget Tr_meulage_motif_1_153 := [[-29.824615234375,-68.797875,83.0298125],[0.61859167979337,-0.623266759536001,0.339563067143743,-0.337016028669028],[0,0,0,0],[8.999999E+09,8.999999E+09,8.999999E+09,8.999999E+09,8.999999E+09,8.999999E+09]];
    LOCAL CONST Robtarget Tr_meulage_motif_1_154 := [[-29.274076171875,-69.6326875,83.0298125],[0.61859167979337,-0.623266759536001,0.339563067143743,-0.337016028669028],[0,0,0,0],[8.999999E+09,8.999999E+09,8.999999E+09,8.999999E+09,8.999999E+09,8.999999E+09]];
    LOCAL CONST Robtarget Tr_meulage_motif_1_155 := [[-28.72353515625,-70.4674921875,83.0298125],[0.61859167979337,-0.623266759536001,0.339563067143743,-0.337016028669028],[0,0,0,0],[8.999999E+09,8.999999E+09,8.999999E+09,8.999999E+09,8.999999E+09,8.999999E+09]];
    LOCAL CONST Robtarget Tr_meulage_motif_1_156 := [[-28.17299609375,-71.3023046875,83.0298125],[0.61859167979337,-0.623266759536001,0.339563067143743,-0.337016028669028],[0,0,0,0],[8.999999E+09,8.999999E+09,8.999999E+09,8.999999E+09,8.999999E+09,8.999999E+09]];
    LOCAL CONST Robtarget Tr_meulage_motif_1_157 := [[-27.622455078125,-72.137109375,83.0298125],[0.61859167979337,-0.623266759536001,0.339563067143743,-0.337016028669028],[0,0,0,0],[8.999999E+09,8.999999E+09,8.999999E+09,8.999999E+09,8.999999E+09,8.999999E+09]];
    LOCAL CONST Robtarget Tr_meulage_motif_1_158 := [[-27.071916015625,-72.971921875,83.0298125],[0.61859167979337,-0.623266759536001,0.339563067143743,-0.337016028669028],[0,0,0,0],[8.999999E+09,8.999999E+09,8.999999E+09,8.999999E+09,8.999999E+09,8.999999E+09]];
    LOCAL CONST Robtarget Tr_meulage_motif_1_159 := [[-26.521375,-73.8067265625,83.0298125],[0.61859167979337,-0.623266759536001,0.339563067143743,-0.337016028669028],[0,0,0,0],[8.999999E+09,8.999999E+09,8.999999E+09,8.999999E+09,8.999999E+09,8.999999E+09]];
    LOCAL CONST Robtarget Tr_meulage_motif_1_160 := [[-25.9708359375,-74.6415390625,83.0298125],[0.61859167979337,-0.623266759536001,0.339563067143743,-0.337016028669028],[0,0,0,0],[8.999999E+09,8.999999E+09,8.999999E+09,8.999999E+09,8.999999E+09,8.999999E+09]];
    LOCAL CONST Robtarget Tr_meulage_motif_1_161 := [[-25.420296875,-75.4763515625,83.0298125],[0.61859167979337,-0.623266759536001,0.339563067143743,-0.337016028669028],[0,0,0,0],[8.999999E+09,8.999999E+09,8.999999E+09,8.999999E+09,8.999999E+09,8.999999E+09]];
    LOCAL CONST Robtarget Tr_meulage_motif_1_162 := [[-24.869755859375,-76.31115625,83.0298125],[0.61859167979337,-0.623266759536001,0.339563067143743,-0.337016028669028],[0,0,0,0],[8.999999E+09,8.999999E+09,8.999999E+09,8.999999E+09,8.999999E+09,8.999999E+09]];
    LOCAL CONST Robtarget Tr_meulage_motif_1_163 := [[-24.319216796875,-77.14596875,83.0298125],[0.61859167979337,-0.623266759536001,0.339563067143743,-0.337016028669028],[0,0,0,0],[8.999999E+09,8.999999E+09,8.999999E+09,8.999999E+09,8.999999E+09,8.999999E+09]];
    LOCAL CONST Robtarget Tr_meulage_motif_1_164 := [[-23.76867578125,-77.9807734375,83.0298125],[0.61859167979337,-0.623266759536001,0.339563067143743,-0.337016028669028],[0,0,0,0],[8.999999E+09,8.999999E+09,8.999999E+09,8.999999E+09,8.999999E+09,8.999999E+09]];
    LOCAL CONST Robtarget Tr_meulage_motif_1_165 := [[-23.21813671875,-78.8155859375,83.0298125],[0.61859167979337,-0.623266759536001,0.339563067143743,-0.337016028669028],[0,0,0,0],[8.999999E+09,8.999999E+09,8.999999E+09,8.999999E+09,8.999999E+09,8.999999E+09]];
    LOCAL CONST Robtarget Tr_meulage_motif_1_166 := [[-22.66759765625,-79.650390625,83.0298125],[0.61859167979337,-0.623266759536001,0.339563067143743,-0.337016028669028],[0,0,0,0],[8.999999E+09,8.999999E+09,8.999999E+09,8.999999E+09,8.999999E+09,8.999999E+09]];
    LOCAL CONST Robtarget Tr_meulage_motif_1_167 := [[-22.117056640625,-80.485203125,83.0298125],[0.61859167979337,-0.623266759536001,0.339563067143743,-0.337016028669028],[0,0,0,0],[8.999999E+09,8.999999E+09,8.999999E+09,8.999999E+09,8.999999E+09,8.999999E+09]];
    LOCAL CONST Robtarget Tr_meulage_motif_1_168 := [[-21.566517578125,-81.3200078125,83.0298125],[0.61859167979337,-0.623266759536001,0.339563067143743,-0.337016028669028],[0,0,0,0],[8.999999E+09,8.999999E+09,8.999999E+09,8.999999E+09,8.999999E+09,8.999999E+09]];
    LOCAL CONST Robtarget Tr_meulage_motif_1_169 := [[-21.0159765625,-82.1548203125,83.0298125],[0.61859167979337,-0.623266759536001,0.339563067143743,-0.337016028669028],[0,0,0,0],[8.999999E+09,8.999999E+09,8.999999E+09,8.999999E+09,8.999999E+09,8.999999E+09]];
    LOCAL CONST Robtarget Tr_meulage_motif_1_170 := [[-20.4654375,-82.989625,83.0298125],[0.61859167979337,-0.623266759536001,0.339563067143743,-0.337016028669028],[0,0,0,0],[8.999999E+09,8.999999E+09,8.999999E+09,8.999999E+09,8.999999E+09,8.999999E+09]];
    LOCAL CONST Robtarget Tr_meulage_motif_1_171 := [[-19.9148984375,-83.8244375,83.0298125],[0.61859167979337,-0.623266759536001,0.339563067143743,-0.337016028669028],[0,0,0,0],[8.999999E+09,8.999999E+09,8.999999E+09,8.999999E+09,8.999999E+09,8.999999E+09]];
    LOCAL CONST Robtarget Tr_meulage_motif_1_172 := [[-19.364357421875,-84.6592421875,83.0298125],[0.61859167979337,-0.623266759536001,0.339563067143743,-0.337016028669028],[0,0,0,0],[8.999999E+09,8.999999E+09,8.999999E+09,8.999999E+09,8.999999E+09,8.999999E+09]];
    LOCAL CONST Robtarget Tr_meulage_motif_1_173 := [[-18.813818359375,-85.4940546875,83.0298125],[0.61859167979337,-0.623266759536001,0.339563067143743,-0.337016028669028],[0,0,0,0],[8.999999E+09,8.999999E+09,8.999999E+09,8.999999E+09,8.999999E+09,8.999999E+09]];
    LOCAL CONST Robtarget Tr_meulage_motif_1_174 := [[-18.26327734375,-86.328859375,83.0298125],[0.61859167979337,-0.623266759536001,0.339563067143743,-0.337016028669028],[0,0,0,0],[8.999999E+09,8.999999E+09,8.999999E+09,8.999999E+09,8.999999E+09,8.999999E+09]];
    LOCAL CONST Robtarget Tr_meulage_motif_1_175 := [[-17.71273828125,-87.163671875,83.0298125],[0.61859167979337,-0.623266759536001,0.339563067143743,-0.337016028669028],[0,0,0,0],[8.999999E+09,8.999999E+09,8.999999E+09,8.999999E+09,8.999999E+09,8.999999E+09]];
    LOCAL CONST Robtarget Tr_meulage_motif_1_176 := [[-17.162197265625,-87.998484375,83.0298125],[0.61859167979337,-0.623266759536001,0.339563067143743,-0.337016028669028],[0,0,0,0],[8.999999E+09,8.999999E+09,8.999999E+09,8.999999E+09,8.999999E+09,8.999999E+09]];
    LOCAL CONST Robtarget Tr_meulage_motif_1_177 := [[-16.611658203125,-88.8332890625,83.0298125],[0.61859167979337,-0.623266759536001,0.339563067143743,-0.337016028669028],[0,0,0,0],[8.999999E+09,8.999999E+09,8.999999E+09,8.999999E+09,8.999999E+09,8.999999E+09]];
    LOCAL CONST Robtarget Tr_meulage_motif_1_178 := [[-16.0611181640625,-89.6681015625,83.0298125],[0.61859167979337,-0.623266759536001,0.339563067143743,-0.337016028669028],[0,0,0,0],[8.999999E+09,8.999999E+09,8.999999E+09,8.999999E+09,8.999999E+09,8.999999E+09]];
    LOCAL CONST Robtarget Tr_meulage_motif_1_179 := [[-15.510578125,-90.50290625,83.0298125],[0.61859167979337,-0.623266759536001,0.339563067143743,-0.337016028669028],[0,0,0,0],[8.999999E+09,8.999999E+09,8.999999E+09,8.999999E+09,8.999999E+09,8.999999E+09]];
    LOCAL CONST Robtarget Tr_meulage_motif_1_180 := [[-14.9600390625,-91.33771875,83.0298125],[0.61859167979337,-0.623266759536001,0.339563067143743,-0.337016028669028],[0,0,0,0],[8.999999E+09,8.999999E+09,8.999999E+09,8.999999E+09,8.999999E+09,8.999999E+09]];
    LOCAL CONST Robtarget Tr_meulage_motif_1_181 := [[-14.4094990234375,-92.1725234375,83.0298125],[0.61859167979337,-0.623266759536001,0.339563067143743,-0.337016028669028],[0,0,0,0],[8.999999E+09,8.999999E+09,8.999999E+09,8.999999E+09,8.999999E+09,8.999999E+09]];
    LOCAL CONST Robtarget Tr_meulage_motif_1_182 := [[-13.858958984375,-93.0073359375,83.0298125],[0.61859167979337,-0.623266759536001,0.339563067143743,-0.337016028669028],[0,0,0,0],[8.999999E+09,8.999999E+09,8.999999E+09,8.999999E+09,8.999999E+09,8.999999E+09]];
    LOCAL CONST Robtarget Tr_meulage_motif_1_183 := [[-13.3084189453125,-93.842140625,83.0298125],[0.61859167979337,-0.623266759536001,0.339563067143743,-0.337016028669028],[0,0,0,0],[8.999999E+09,8.999999E+09,8.999999E+09,8.999999E+09,8.999999E+09,8.999999E+09]];
    LOCAL CONST Robtarget Tr_meulage_motif_1_184 := [[-12.75787890625,-94.676953125,83.0298125],[0.61859167979337,-0.623266759536001,0.339563067143743,-0.337016028669028],[0,0,0,0],[8.999999E+09,8.999999E+09,8.999999E+09,8.999999E+09,8.999999E+09,8.999999E+09]];
    LOCAL CONST Robtarget Tr_meulage_motif_1_185 := [[-12.2073388671875,-95.5117578125,83.0298125],[0.61859167979337,-0.623266759536001,0.339563067143743,-0.337016028669028],[0,0,0,0],[8.999999E+09,8.999999E+09,8.999999E+09,8.999999E+09,8.999999E+09,8.999999E+09]];
    LOCAL CONST Robtarget Tr_meulage_motif_1_186 := [[-11.6567998046875,-96.3465703125,83.0298125],[0.61859167979337,-0.623266759536001,0.339563067143743,-0.337016028669028],[0,0,0,0],[8.999999E+09,8.999999E+09,8.999999E+09,8.999999E+09,8.999999E+09,8.999999E+09]];
    LOCAL CONST Robtarget Tr_meulage_motif_1_187 := [[-11.106259765625,-97.181375,83.0298125],[0.61859167979337,-0.623266759536001,0.339563067143743,-0.337016028669028],[0,0,0,0],[8.999999E+09,8.999999E+09,8.999999E+09,8.999999E+09,8.999999E+09,8.999999E+09]];
    LOCAL CONST Robtarget Tr_meulage_motif_1_188 := [[-10.5557197265625,-98.0161875,83.0298125],[0.61859167979337,-0.623266759536001,0.339563067143743,-0.337016028669028],[0,0,0,0],[8.999999E+09,8.999999E+09,8.999999E+09,8.999999E+09,8.999999E+09,8.999999E+09]];
    LOCAL CONST Robtarget Tr_meulage_motif_1_189 := [[-10.0093916015625,-98.8448671875,82.91921875],[0.61859167979337,-0.623266759536001,0.339563067143743,-0.337016028669028],[0,0,0,0],[8.999999E+09,8.999999E+09,8.999999E+09,8.999999E+09,8.999999E+09,8.999999E+09]];
    LOCAL CONST Robtarget Tr_meulage_motif_1_190 := [[-9.488529296875,-99.63515625,82.70803125],[0.61859167979337,-0.623266759536001,0.339563067143743,-0.337016028669028],[0,0,0,0],[8.999999E+09,8.999999E+09,8.999999E+09,8.999999E+09,8.999999E+09,8.999999E+09]];
    LOCAL CONST Robtarget Tr_meulage_motif_1_191 := [[-9.019361328125,-100.347203125,82.4361875],[0.61859167979337,-0.623266759536001,0.339563067143743,-0.337016028669028],[0,0,0,0],[8.999999E+09,8.999999E+09,8.999999E+09,8.999999E+09,8.999999E+09,8.999999E+09]];
    LOCAL CONST Robtarget Tr_meulage_motif_1_192 := [[-8.606783203125,-100.973453125,82.16025],[0.61859167979337,-0.623266759536001,0.339563067143743,-0.337016028669028],[0,0,0,0],[8.999999E+09,8.999999E+09,8.999999E+09,8.999999E+09,8.999999E+09,8.999999E+09]];
    LOCAL CONST Robtarget Tr_meulage_motif_1_193 := [[-8.00125732421875,-101.8930625,81.5441328125],[0.61859167979337,-0.623266759536001,0.339563067143743,-0.337016028669028],[0,0,0,0],[8.999999E+09,8.999999E+09,8.999999E+09,8.999999E+09,8.999999E+09,8.999999E+09]];
    LOCAL CONST Robtarget Tr_meulage_motif_1_194 := [[-7.43847119140625,-102.748390625,80.6964765625],[0.61859167979337,-0.623266759536001,0.339563067143743,-0.337016028669028],[0,0,0,0],[8.999999E+09,8.999999E+09,8.999999E+09,8.999999E+09,8.999999E+09,8.999999E+09]];
    LOCAL CONST Robtarget Tr_meulage_motif_1_195 := [[-6.97288720703125,-103.4567421875,79.6726015625],[0.61859167979337,-0.623266759536001,0.339563067143743,-0.337016028669028],[0,0,0,0],[8.999999E+09,8.999999E+09,8.999999E+09,8.999999E+09,8.999999E+09,8.999999E+09]];
    LOCAL CONST Robtarget Tr_meulage_motif_1_196 := [[-6.7053203125,-103.8650390625,78.5564140625],[0.61859167979337,-0.623266759536001,0.339563067143743,-0.337016028669028],[0,0,0,0],[8.999999E+09,8.999999E+09,8.999999E+09,8.999999E+09,8.999999E+09,8.999999E+09]];
    LOCAL CONST Robtarget Tr_meulage_motif_1_197 := [[-6.691158203125,-103.8881171875,77.8604453125],[0.61859167979337,-0.623266759536001,0.339563067143743,-0.337016028669028],[0,0,0,0],[8.999999E+09,8.999999E+09,8.999999E+09,8.999999E+09,8.999999E+09,8.999999E+09]];
    LOCAL CONST Robtarget Tr_meulage_motif_1_198 := [[-6.69185888671875,-103.888578125,77.1991953125],[0.61859167979337,-0.623266759536001,0.339563067143743,-0.337016028669028],[0,0,0,0],[8.999999E+09,8.999999E+09,8.999999E+09,8.999999E+09,8.999999E+09,8.999999E+09]];
    LOCAL CONST Robtarget Tr_meulage_motif_1_199 := [[-6.72277001953125,-103.8432265625,76.5381015625],[0.61859167979337,-0.623266759536001,0.339563067143743,-0.337016028669028],[0,0,0,0],[8.999999E+09,8.999999E+09,8.999999E+09,8.999999E+09,8.999999E+09,8.999999E+09]];
    LOCAL CONST Robtarget Tr_meulage_motif_1_200 := [[-6.9982265625,-103.428078125,75.4363515625],[0.61859167979337,-0.623266759536001,0.339563067143743,-0.337016028669028],[0,0,0,0],[8.999999E+09,8.999999E+09,8.999999E+09,8.999999E+09,8.999999E+09,8.999999E+09]];
    LOCAL CONST Robtarget Tr_meulage_motif_1_201 := [[-7.47089892578125,-102.7136640625,74.4297265625],[0.61859167979337,-0.623266759536001,0.339563067143743,-0.337016028669028],[0,0,0,0],[8.999999E+09,8.999999E+09,8.999999E+09,8.999999E+09,8.999999E+09,8.999999E+09]];
    LOCAL CONST Robtarget Tr_meulage_motif_1_202 := [[-8.03522021484375,-101.8598671875,73.6008515625],[0.61859167979337,-0.623266759536001,0.339563067143743,-0.337016028669028],[0,0,0,0],[8.999999E+09,8.999999E+09,8.999999E+09,8.999999E+09,8.999999E+09,8.999999E+09]];
    LOCAL CONST Robtarget Tr_meulage_motif_1_203 := [[-8.41389453125,-101.286578125,73.2051015625],[0.61859167979337,-0.623266759536001,0.339563067143743,-0.337016028669028],[0,0,0,0],[8.999999E+09,8.999999E+09,8.999999E+09,8.999999E+09,8.999999E+09,8.999999E+09]];
    LOCAL CONST Robtarget Tr_meulage_motif_1_204 := [[-9.0520224609375,-100.3200859375,72.7175703125],[0.61859167979337,-0.623266759536001,0.339563067143743,-0.337016028669028],[0,0,0,0],[8.999999E+09,8.999999E+09,8.999999E+09,8.999999E+09,8.999999E+09,8.999999E+09]];
    LOCAL CONST Robtarget Tr_meulage_motif_1_205 := [[-9.517525390625,-99.614828125,72.4534765625],[0.61859167979337,-0.623266759536001,0.339563067143743,-0.337016028669028],[0,0,0,0],[8.999999E+09,8.999999E+09,8.999999E+09,8.999999E+09,8.999999E+09,8.999999E+09]];
    LOCAL CONST Robtarget Tr_meulage_motif_1_206 := [[-10.0308447265625,-98.8369296875,72.2490078125],[0.61859167979337,-0.623266759536001,0.339563067143743,-0.337016028669028],[0,0,0,0],[8.999999E+09,8.999999E+09,8.999999E+09,8.999999E+09,8.999999E+09,8.999999E+09]];
    LOCAL CONST Robtarget Tr_meulage_motif_1_207 := [[-10.571349609375,-98.0175859375,72.1404140625],[0.61859167979337,-0.623266759536001,0.339563067143743,-0.337016028669028],[0,0,0,0],[8.999999E+09,8.999999E+09,8.999999E+09,8.999999E+09,8.999999E+09,8.999999E+09]];
    LOCAL CONST Robtarget Tr_meulage_motif_1_208 := [[-11.117912109375,-97.1890625,72.0298203125],[0.61859167979337,-0.623266759536001,0.339563067143743,-0.337016028669028],[0,0,0,0],[8.999999E+09,8.999999E+09,8.999999E+09,8.999999E+09,8.999999E+09,8.999999E+09]];
    LOCAL CONST Robtarget Tr_meulage_motif_1_209 := [[-11.6684521484375,-96.3542578125,72.0298203125],[0.61859167979337,-0.623266759536001,0.339563067143743,-0.337016028669028],[0,0,0,0],[8.999999E+09,8.999999E+09,8.999999E+09,8.999999E+09,8.999999E+09,8.999999E+09]];
    LOCAL CONST Robtarget Tr_meulage_motif_1_210 := [[-12.2189912109375,-95.5194453125,72.0298203125],[0.61859167979337,-0.623266759536001,0.339563067143743,-0.337016028669028],[0,0,0,0],[8.999999E+09,8.999999E+09,8.999999E+09,8.999999E+09,8.999999E+09,8.999999E+09]];
    LOCAL CONST Robtarget Tr_meulage_motif_1_211 := [[-12.76953125,-94.684640625,72.0298203125],[0.61859167979337,-0.623266759536001,0.339563067143743,-0.337016028669028],[0,0,0,0],[8.999999E+09,8.999999E+09,8.999999E+09,8.999999E+09,8.999999E+09,8.999999E+09]];
    LOCAL CONST Robtarget Tr_meulage_motif_1_212 := [[-13.3200712890625,-93.849828125,72.0298203125],[0.61859167979337,-0.623266759536001,0.339563067143743,-0.337016028669028],[0,0,0,0],[8.999999E+09,8.999999E+09,8.999999E+09,8.999999E+09,8.999999E+09,8.999999E+09]];
    LOCAL CONST Robtarget Tr_meulage_motif_1_213 := [[-13.870611328125,-93.0150234375,72.0298203125],[0.61859167979337,-0.623266759536001,0.339563067143743,-0.337016028669028],[0,0,0,0],[8.999999E+09,8.999999E+09,8.999999E+09,8.999999E+09,8.999999E+09,8.999999E+09]];
    LOCAL CONST Robtarget Tr_meulage_motif_1_214 := [[-14.4211513671875,-92.1802109375,72.0298203125],[0.61859167979337,-0.623266759536001,0.339563067143743,-0.337016028669028],[0,0,0,0],[8.999999E+09,8.999999E+09,8.999999E+09,8.999999E+09,8.999999E+09,8.999999E+09]];
    LOCAL CONST Robtarget Tr_meulage_motif_1_215 := [[-14.97169140625,-91.34540625,72.0298203125],[0.61859167979337,-0.623266759536001,0.339563067143743,-0.337016028669028],[0,0,0,0],[8.999999E+09,8.999999E+09,8.999999E+09,8.999999E+09,8.999999E+09,8.999999E+09]];
    LOCAL CONST Robtarget Tr_meulage_motif_1_216 := [[-15.52223046875,-90.51059375,72.0298203125],[0.61859167979337,-0.623266759536001,0.339563067143743,-0.337016028669028],[0,0,0,0],[8.999999E+09,8.999999E+09,8.999999E+09,8.999999E+09,8.999999E+09,8.999999E+09]];
    LOCAL CONST Robtarget Tr_meulage_motif_1_217 := [[-16.0727705078125,-89.67578125,72.0298203125],[0.61859167979337,-0.623266759536001,0.339563067143743,-0.337016028669028],[0,0,0,0],[8.999999E+09,8.999999E+09,8.999999E+09,8.999999E+09,8.999999E+09,8.999999E+09]];
    LOCAL CONST Robtarget Tr_meulage_motif_1_218 := [[-16.623310546875,-88.8409765625,72.0298203125],[0.61859167979337,-0.623266759536001,0.339563067143743,-0.337016028669028],[0,0,0,0],[8.999999E+09,8.999999E+09,8.999999E+09,8.999999E+09,8.999999E+09,8.999999E+09]];
    LOCAL CONST Robtarget Tr_meulage_motif_1_219 := [[-17.173849609375,-88.0061640625,72.0298203125],[0.61859167979337,-0.623266759536001,0.339563067143743,-0.337016028669028],[0,0,0,0],[8.999999E+09,8.999999E+09,8.999999E+09,8.999999E+09,8.999999E+09,8.999999E+09]];
    LOCAL CONST Robtarget Tr_meulage_motif_1_220 := [[-17.724390625,-87.171359375,72.0298203125],[0.61859167979337,-0.623266759536001,0.339563067143743,-0.337016028669028],[0,0,0,0],[8.999999E+09,8.999999E+09,8.999999E+09,8.999999E+09,8.999999E+09,8.999999E+09]];
    LOCAL CONST Robtarget Tr_meulage_motif_1_221 := [[-18.2749296875,-86.336546875,72.0298203125],[0.61859167979337,-0.623266759536001,0.339563067143743,-0.337016028669028],[0,0,0,0],[8.999999E+09,8.999999E+09,8.999999E+09,8.999999E+09,8.999999E+09,8.999999E+09]];
    LOCAL CONST Robtarget Tr_meulage_motif_1_222 := [[-18.825470703125,-85.5017421875,72.0298203125],[0.61859167979337,-0.623266759536001,0.339563067143743,-0.337016028669028],[0,0,0,0],[8.999999E+09,8.999999E+09,8.999999E+09,8.999999E+09,8.999999E+09,8.999999E+09]];
    LOCAL CONST Robtarget Tr_meulage_motif_1_223 := [[-19.376009765625,-84.6669296875,72.0298203125],[0.61859167979337,-0.623266759536001,0.339563067143743,-0.337016028669028],[0,0,0,0],[8.999999E+09,8.999999E+09,8.999999E+09,8.999999E+09,8.999999E+09,8.999999E+09]];
    LOCAL CONST Robtarget Tr_meulage_motif_1_224 := [[-19.926548828125,-83.832125,72.0298203125],[0.61859167979337,-0.623266759536001,0.339563067143743,-0.337016028669028],[0,0,0,0],[8.999999E+09,8.999999E+09,8.999999E+09,8.999999E+09,8.999999E+09,8.999999E+09]];
    LOCAL CONST Robtarget Tr_meulage_motif_1_225 := [[-20.47708984375,-82.9973125,72.0298203125],[0.61859167979337,-0.623266759536001,0.339563067143743,-0.337016028669028],[0,0,0,0],[8.999999E+09,8.999999E+09,8.999999E+09,8.999999E+09,8.999999E+09,8.999999E+09]];
    LOCAL CONST Robtarget Tr_meulage_motif_1_226 := [[-21.02762890625,-82.1625078125,72.0298203125],[0.61859167979337,-0.623266759536001,0.339563067143743,-0.337016028669028],[0,0,0,0],[8.999999E+09,8.999999E+09,8.999999E+09,8.999999E+09,8.999999E+09,8.999999E+09]];
    LOCAL CONST Robtarget Tr_meulage_motif_1_227 := [[-21.578169921875,-81.3276953125,72.0298203125],[0.61859167979337,-0.623266759536001,0.339563067143743,-0.337016028669028],[0,0,0,0],[8.999999E+09,8.999999E+09,8.999999E+09,8.999999E+09,8.999999E+09,8.999999E+09]];
    LOCAL CONST Robtarget Tr_meulage_motif_1_228 := [[-22.128708984375,-80.492890625,72.0298203125],[0.61859167979337,-0.623266759536001,0.339563067143743,-0.337016028669028],[0,0,0,0],[8.999999E+09,8.999999E+09,8.999999E+09,8.999999E+09,8.999999E+09,8.999999E+09]];
    LOCAL CONST Robtarget Tr_meulage_motif_1_229 := [[-22.67925,-79.658078125,72.0298203125],[0.61859167979337,-0.623266759536001,0.339563067143743,-0.337016028669028],[0,0,0,0],[8.999999E+09,8.999999E+09,8.999999E+09,8.999999E+09,8.999999E+09,8.999999E+09]];
    LOCAL CONST Robtarget Tr_meulage_motif_1_230 := [[-23.2297890625,-78.823265625,72.0298203125],[0.61859167979337,-0.623266759536001,0.339563067143743,-0.337016028669028],[0,0,0,0],[8.999999E+09,8.999999E+09,8.999999E+09,8.999999E+09,8.999999E+09,8.999999E+09]];
    LOCAL CONST Robtarget Tr_meulage_motif_1_231 := [[-23.780328125,-77.9884609375,72.0298203125],[0.61859167979337,-0.623266759536001,0.339563067143743,-0.337016028669028],[0,0,0,0],[8.999999E+09,8.999999E+09,8.999999E+09,8.999999E+09,8.999999E+09,8.999999E+09]];
    LOCAL CONST Robtarget Tr_meulage_motif_1_232 := [[-24.330869140625,-77.1536484375,72.0298203125],[0.61859167979337,-0.623266759536001,0.339563067143743,-0.337016028669028],[0,0,0,0],[8.999999E+09,8.999999E+09,8.999999E+09,8.999999E+09,8.999999E+09,8.999999E+09]];
    LOCAL CONST Robtarget Tr_meulage_motif_1_233 := [[-24.881408203125,-76.31884375,72.0298203125],[0.61859167979337,-0.623266759536001,0.339563067143743,-0.337016028669028],[0,0,0,0],[8.999999E+09,8.999999E+09,8.999999E+09,8.999999E+09,8.999999E+09,8.999999E+09]];
    LOCAL CONST Robtarget Tr_meulage_motif_1_234 := [[-25.43194921875,-75.48403125,72.0298203125],[0.61859167979337,-0.623266759536001,0.339563067143743,-0.337016028669028],[0,0,0,0],[8.999999E+09,8.999999E+09,8.999999E+09,8.999999E+09,8.999999E+09,8.999999E+09]];
    LOCAL CONST Robtarget Tr_meulage_motif_1_235 := [[-25.98248828125,-74.6492265625,72.0298203125],[0.61859167979337,-0.623266759536001,0.339563067143743,-0.337016028669028],[0,0,0,0],[8.999999E+09,8.999999E+09,8.999999E+09,8.999999E+09,8.999999E+09,8.999999E+09]];
    LOCAL CONST Robtarget Tr_meulage_motif_1_236 := [[-26.53302734375,-73.8144140625,72.0298203125],[0.61859167979337,-0.623266759536001,0.339563067143743,-0.337016028669028],[0,0,0,0],[8.999999E+09,8.999999E+09,8.999999E+09,8.999999E+09,8.999999E+09,8.999999E+09]];
    LOCAL CONST Robtarget Tr_meulage_motif_1_237 := [[-27.083568359375,-72.979609375,72.0298203125],[0.61859167979337,-0.623266759536001,0.339563067143743,-0.337016028669028],[0,0,0,0],[8.999999E+09,8.999999E+09,8.999999E+09,8.999999E+09,8.999999E+09,8.999999E+09]];
    LOCAL CONST Robtarget Tr_meulage_motif_1_238 := [[-27.634107421875,-72.144796875,72.0298203125],[0.61859167979337,-0.623266759536001,0.339563067143743,-0.337016028669028],[0,0,0,0],[8.999999E+09,8.999999E+09,8.999999E+09,8.999999E+09,8.999999E+09,8.999999E+09]];
    LOCAL CONST Robtarget Tr_meulage_motif_1_239 := [[-28.1846484375,-71.3099921875,72.0298203125],[0.61859167979337,-0.623266759536001,0.339563067143743,-0.337016028669028],[0,0,0,0],[8.999999E+09,8.999999E+09,8.999999E+09,8.999999E+09,8.999999E+09,8.999999E+09]];
    LOCAL CONST Robtarget Tr_meulage_motif_1_240 := [[-28.7351875,-70.4751796875,72.0298203125],[0.61859167979337,-0.623266759536001,0.339563067143743,-0.337016028669028],[0,0,0,0],[8.999999E+09,8.999999E+09,8.999999E+09,8.999999E+09,8.999999E+09,8.999999E+09]];
    LOCAL CONST Robtarget Tr_meulage_motif_1_241 := [[-29.285728515625,-69.640375,72.0298203125],[0.61859167979337,-0.623266759536001,0.339563067143743,-0.337016028669028],[0,0,0,0],[8.999999E+09,8.999999E+09,8.999999E+09,8.999999E+09,8.999999E+09,8.999999E+09]];
    LOCAL CONST Robtarget Tr_meulage_motif_1_242 := [[-29.836267578125,-68.8055625,72.0298203125],[0.61859167979337,-0.623266759536001,0.339563067143743,-0.337016028669028],[0,0,0,0],[8.999999E+09,8.999999E+09,8.999999E+09,8.999999E+09,8.999999E+09,8.999999E+09]];
    LOCAL CONST Robtarget Tr_meulage_motif_1_243 := [[-30.386806640625,-67.9707578125,72.0298203125],[0.61859167979337,-0.623266759536001,0.339563067143743,-0.337016028669028],[0,0,0,0],[8.999999E+09,8.999999E+09,8.999999E+09,8.999999E+09,8.999999E+09,8.999999E+09]];
    LOCAL CONST Robtarget Tr_meulage_motif_1_244 := [[-30.93734765625,-67.1359453125,72.0298203125],[0.61859167979337,-0.623266759536001,0.339563067143743,-0.337016028669028],[0,0,0,0],[8.999999E+09,8.999999E+09,8.999999E+09,8.999999E+09,8.999999E+09,8.999999E+09]];
    LOCAL CONST Robtarget Tr_meulage_motif_1_245 := [[-31.48788671875,-66.3011328125,72.0298203125],[0.61859167979337,-0.623266759536001,0.339563067143743,-0.337016028669028],[0,0,0,0],[8.999999E+09,8.999999E+09,8.999999E+09,8.999999E+09,8.999999E+09,8.999999E+09]];
    LOCAL CONST Robtarget Tr_meulage_motif_1_246 := [[-32.038427734375,-65.466328125,72.0298203125],[0.61859167979337,-0.623266759536001,0.339563067143743,-0.337016028669028],[0,0,0,0],[8.999999E+09,8.999999E+09,8.999999E+09,8.999999E+09,8.999999E+09,8.999999E+09]];
    LOCAL CONST Robtarget Tr_meulage_motif_1_247 := [[-32.588966796875,-64.63151953125,72.0298203125],[0.61859167979337,-0.623266759536001,0.339563067143743,-0.337016028669028],[0,0,0,0],[8.999999E+09,8.999999E+09,8.999999E+09,8.999999E+09,8.999999E+09,8.999999E+09]];
    LOCAL CONST Robtarget Tr_meulage_motif_1_248 := [[-33.1395078125,-63.7967109375,72.0298203125],[0.61859167979337,-0.623266759536001,0.339563067143743,-0.337016028669028],[0,0,0,0],[8.999999E+09,8.999999E+09,8.999999E+09,8.999999E+09,8.999999E+09,8.999999E+09]];
    LOCAL CONST Robtarget Tr_meulage_motif_1_249 := [[-33.690046875,-62.96190234375,72.0298203125],[0.61859167979337,-0.623266759536001,0.339563067143743,-0.337016028669028],[0,0,0,0],[8.999999E+09,8.999999E+09,8.999999E+09,8.999999E+09,8.999999E+09,8.999999E+09]];
    LOCAL CONST Robtarget Tr_meulage_motif_1_250 := [[-34.2405859375,-62.12709375,72.0298203125],[0.61859167979337,-0.623266759536001,0.339563067143743,-0.337016028669028],[0,0,0,0],[8.999999E+09,8.999999E+09,8.999999E+09,8.999999E+09,8.999999E+09,8.999999E+09]];
    LOCAL CONST Robtarget Tr_meulage_motif_1_251 := [[-34.791125,-61.29228125,72.0298203125],[0.61859167979337,-0.623266759536001,0.339563067143743,-0.337016028669028],[0,0,0,0],[8.999999E+09,8.999999E+09,8.999999E+09,8.999999E+09,8.999999E+09,8.999999E+09]];
    LOCAL CONST Robtarget Tr_meulage_motif_1_252 := [[-35.34166796875,-60.45747265625,72.0298203125],[0.61859167979337,-0.623266759536001,0.339563067143743,-0.337016028669028],[0,0,0,0],[8.999999E+09,8.999999E+09,8.999999E+09,8.999999E+09,8.999999E+09,8.999999E+09]];
    LOCAL CONST Robtarget Tr_meulage_motif_1_253 := [[-35.89220703125,-59.6226640625,72.0298203125],[0.61859167979337,-0.623266759536001,0.339563067143743,-0.337016028669028],[0,0,0,0],[8.999999E+09,8.999999E+09,8.999999E+09,8.999999E+09,8.999999E+09,8.999999E+09]];
    LOCAL CONST Robtarget Tr_meulage_motif_1_254 := [[-36.44274609375,-58.78785546875,72.0298203125],[0.61859167979337,-0.623266759536001,0.339563067143743,-0.337016028669028],[0,0,0,0],[8.999999E+09,8.999999E+09,8.999999E+09,8.999999E+09,8.999999E+09,8.999999E+09]];
    LOCAL CONST Robtarget Tr_meulage_motif_1_255 := [[-36.99328515625,-57.953046875,72.0298203125],[0.61859167979337,-0.623266759536001,0.339563067143743,-0.337016028669028],[0,0,0,0],[8.999999E+09,8.999999E+09,8.999999E+09,8.999999E+09,8.999999E+09,8.999999E+09]];
    LOCAL CONST Robtarget Tr_meulage_motif_1_256 := [[-37.53984765625,-57.1245234375,71.9192265625],[0.61859167979337,-0.623266759536001,0.339563067143743,-0.337016028669028],[0,0,0,0],[8.999999E+09,8.999999E+09,8.999999E+09,8.999999E+09,8.999999E+09,8.999999E+09]];
    LOCAL CONST Robtarget Tr_meulage_motif_1_257 := [[-38.06115625,-56.33452734375,71.7080390625],[0.61859167979337,-0.623266759536001,0.339563067143743,-0.337016028669028],[0,0,0,0],[8.999999E+09,8.999999E+09,8.999999E+09,8.999999E+09,8.999999E+09,8.999999E+09]];
    LOCAL CONST Robtarget Tr_meulage_motif_1_258 := [[-38.53090234375,-55.622859375,71.4361953125],[0.61859167979337,-0.623266759536001,0.339563067143743,-0.337016028669028],[0,0,0,0],[8.999999E+09,8.999999E+09,8.999999E+09,8.999999E+09,8.999999E+09,8.999999E+09]];
    LOCAL CONST Robtarget Tr_meulage_motif_1_259 := [[-38.92293359375,-55.02910546875,71.1320546875],[0.61859167979337,-0.623266759536001,0.339563067143743,-0.337016028669028],[0,0,0,0],[8.999999E+09,8.999999E+09,8.999999E+09,8.999999E+09,8.999999E+09,8.999999E+09]];
    LOCAL CONST Robtarget Tr_meulage_motif_1_260 := [[-39.49315234375,-54.165984375,70.4695234375],[0.61859167979337,-0.623266759536001,0.339563067143743,-0.337016028669028],[0,0,0,0],[8.999999E+09,8.999999E+09,8.999999E+09,8.999999E+09,8.999999E+09,8.999999E+09]];
    LOCAL CONST Robtarget Tr_meulage_motif_1_261 := [[-39.99066015625,-53.41366796875,69.5675703125],[0.61859167979337,-0.623266759536001,0.339563067143743,-0.337016028669028],[0,0,0,0],[8.999999E+09,8.999999E+09,8.999999E+09,8.999999E+09,8.999999E+09,8.999999E+09]];
    LOCAL CONST Robtarget Tr_meulage_motif_1_262 := [[-40.2862890625,-52.9678046875,68.5215546875],[0.61859167979337,-0.623266759536001,0.339563067143743,-0.337016028669028],[0,0,0,0],[8.999999E+09,8.999999E+09,8.999999E+09,8.999999E+09,8.999999E+09,8.999999E+09]];
    LOCAL CONST Robtarget Tr_meulage_motif_1_263 := [[-40.38875390625,-52.81403125,67.8283203125],[0.61859167979337,-0.623266759536001,0.339563067143743,-0.337016028669028],[0,0,0,0],[8.999999E+09,8.999999E+09,8.999999E+09,8.999999E+09,8.999999E+09,8.999999E+09]];
    LOCAL CONST Robtarget Tr_meulage_motif_1_264 := [[-40.42471484375,-52.76126953125,67.0583203125],[0.61859167979337,-0.623266759536001,0.339563067143743,-0.337016028669028],[0,0,0,0],[8.999999E+09,8.999999E+09,8.999999E+09,8.999999E+09,8.999999E+09,8.999999E+09]];
    LOCAL CONST Robtarget Tr_meulage_motif_1_265 := [[-40.3886796875,-52.8176875,66.2884609375],[0.61859167979337,-0.623266759536001,0.339563067143743,-0.337016028669028],[0,0,0,0],[8.999999E+09,8.999999E+09,8.999999E+09,8.999999E+09,8.999999E+09,8.999999E+09]];
    LOCAL CONST Robtarget Tr_meulage_motif_1_266 := [[-40.1588515625,-53.1687421875,65.18021484375],[0.61859167979337,-0.623266759536001,0.339563067143743,-0.337016028669028],[0,0,0,0],[8.999999E+09,8.999999E+09,8.999999E+09,8.999999E+09,8.999999E+09,8.999999E+09]];
    LOCAL CONST Robtarget Tr_meulage_motif_1_267 := [[-39.931375,-53.5150234375,64.59452734375],[0.61859167979337,-0.623266759536001,0.339563067143743,-0.337016028669028],[0,0,0,0],[8.999999E+09,8.999999E+09,8.999999E+09,8.999999E+09,8.999999E+09,8.999999E+09]];
    LOCAL CONST Robtarget Tr_meulage_motif_1_268 := [[-39.44391796875,-54.25622265625,63.70737109375],[0.61859167979337,-0.623266759536001,0.339563067143743,-0.337016028669028],[0,0,0,0],[8.999999E+09,8.999999E+09,8.999999E+09,8.999999E+09,8.999999E+09,8.999999E+09]];
    LOCAL CONST Robtarget Tr_meulage_motif_1_269 := [[-39.1219140625,-54.74544921875,63.29308984375],[0.61859167979337,-0.623266759536001,0.339563067143743,-0.337016028669028],[0,0,0,0],[8.999999E+09,8.999999E+09,8.999999E+09,8.999999E+09,8.999999E+09,8.999999E+09]];
    LOCAL CONST Robtarget Tr_meulage_motif_1_270 := [[-38.50703515625,-55.6790703125,62.74896484375],[0.61859167979337,-0.623266759536001,0.339563067143743,-0.337016028669028],[0,0,0,0],[8.999999E+09,8.999999E+09,8.999999E+09,8.999999E+09,8.999999E+09,8.999999E+09]];
    LOCAL CONST Robtarget Tr_meulage_motif_1_271 := [[-38.052828125,-56.36848828125,62.45346484375],[0.61859167979337,-0.623266759536001,0.339563067143743,-0.337016028669028],[0,0,0,0],[8.999999E+09,8.999999E+09,8.999999E+09,8.999999E+09,8.999999E+09,8.999999E+09]];
    LOCAL CONST Robtarget Tr_meulage_motif_1_272 := [[-37.53994140625,-57.146671875,62.24898046875],[0.61859167979337,-0.623266759536001,0.339563067143743,-0.337016028669028],[0,0,0,0],[8.999999E+09,8.999999E+09,8.999999E+09,8.999999E+09,8.999999E+09,8.999999E+09]];
    LOCAL CONST Robtarget Tr_meulage_motif_1_273 := [[-36.99966796875,-57.96616796875,62.14043359375],[0.61859167979337,-0.623266759536001,0.339563067143743,-0.337016028669028],[0,0,0,0],[8.999999E+09,8.999999E+09,8.999999E+09,8.999999E+09,8.999999E+09,8.999999E+09]];
    LOCAL CONST Robtarget Tr_meulage_motif_1_274 := [[-36.45333984375,-58.79484375,62.02982421875],[0.61859167979337,-0.623266759536001,0.339563067143743,-0.337016028669028],[0,0,0,0],[8.999999E+09,8.999999E+09,8.999999E+09,8.999999E+09,8.999999E+09,8.999999E+09]];
    LOCAL CONST Robtarget Tr_meulage_motif_1_275 := [[-35.90280078125,-59.62965234375,62.02982421875],[0.61859167979337,-0.623266759536001,0.339563067143743,-0.337016028669028],[0,0,0,0],[8.999999E+09,8.999999E+09,8.999999E+09,8.999999E+09,8.999999E+09,8.999999E+09]];
    LOCAL CONST Robtarget Tr_meulage_motif_1_276 := [[-35.3522578125,-60.4644609375,62.029828125],[0.61859167979337,-0.623266759536001,0.339563067143743,-0.337016028669028],[0,0,0,0],[8.999999E+09,8.999999E+09,8.999999E+09,8.999999E+09,8.999999E+09,8.999999E+09]];
    LOCAL CONST Robtarget Tr_meulage_motif_1_277 := [[-34.80171875,-61.29926953125,62.029828125],[0.61859167979337,-0.623266759536001,0.339563067143743,-0.337016028669028],[0,0,0,0],[8.999999E+09,8.999999E+09,8.999999E+09,8.999999E+09,8.999999E+09,8.999999E+09]];
    LOCAL CONST Robtarget Tr_meulage_motif_1_278 := [[-34.2511796875,-62.134078125,62.029828125],[0.61859167979337,-0.623266759536001,0.339563067143743,-0.337016028669028],[0,0,0,0],[8.999999E+09,8.999999E+09,8.999999E+09,8.999999E+09,8.999999E+09,8.999999E+09]];
    LOCAL CONST Robtarget Tr_meulage_motif_1_279 := [[-33.700640625,-62.96888671875,62.029828125],[0.61859167979337,-0.623266759536001,0.339563067143743,-0.337016028669028],[0,0,0,0],[8.999999E+09,8.999999E+09,8.999999E+09,8.999999E+09,8.999999E+09,8.999999E+09]];
    LOCAL CONST Robtarget Tr_meulage_motif_1_280 := [[-33.1501015625,-63.8036953125,62.029828125],[0.61859167979337,-0.623266759536001,0.339563067143743,-0.337016028669028],[0,0,0,0],[8.999999E+09,8.999999E+09,8.999999E+09,8.999999E+09,8.999999E+09,8.999999E+09]];
    LOCAL CONST Robtarget Tr_meulage_motif_1_281 := [[-32.599560546875,-64.6385078125,62.029828125],[0.61859167979337,-0.623266759536001,0.339563067143743,-0.337016028669028],[0,0,0,0],[8.999999E+09,8.999999E+09,8.999999E+09,8.999999E+09,8.999999E+09,8.999999E+09]];
    LOCAL CONST Robtarget Tr_meulage_motif_1_282 := [[-32.04901953125,-65.47331640625,62.029828125],[0.61859167979337,-0.623266759536001,0.339563067143743,-0.337016028669028],[0,0,0,0],[8.999999E+09,8.999999E+09,8.999999E+09,8.999999E+09,8.999999E+09,8.999999E+09]];
    LOCAL CONST Robtarget Tr_meulage_motif_1_283 := [[-31.49848046875,-66.308125,62.029828125],[0.61859167979337,-0.623266759536001,0.339563067143743,-0.337016028669028],[0,0,0,0],[8.999999E+09,8.999999E+09,8.999999E+09,8.999999E+09,8.999999E+09,8.999999E+09]];
    LOCAL CONST Robtarget Tr_meulage_motif_1_284 := [[-30.947939453125,-67.1429296875,62.029828125],[0.61859167979337,-0.623266759536001,0.339563067143743,-0.337016028669028],[0,0,0,0],[8.999999E+09,8.999999E+09,8.999999E+09,8.999999E+09,8.999999E+09,8.999999E+09]];
    LOCAL CONST Robtarget Tr_meulage_motif_1_285 := [[-30.397400390625,-67.9777421875,62.029828125],[0.61859167979337,-0.623266759536001,0.339563067143743,-0.337016028669028],[0,0,0,0],[8.999999E+09,8.999999E+09,8.999999E+09,8.999999E+09,8.999999E+09,8.999999E+09]];
    LOCAL CONST Robtarget Tr_meulage_motif_1_286 := [[-29.846861328125,-68.812546875,62.029828125],[0.61859167979337,-0.623266759536001,0.339563067143743,-0.337016028669028],[0,0,0,0],[8.999999E+09,8.999999E+09,8.999999E+09,8.999999E+09,8.999999E+09,8.999999E+09]];
    LOCAL CONST Robtarget Tr_meulage_motif_1_287 := [[-29.2963203125,-69.647359375,62.029828125],[0.61859167979337,-0.623266759536001,0.339563067143743,-0.337016028669028],[0,0,0,0],[8.999999E+09,8.999999E+09,8.999999E+09,8.999999E+09,8.999999E+09,8.999999E+09]];
    LOCAL CONST Robtarget Tr_meulage_motif_1_288 := [[-28.74578125,-70.482171875,62.029828125],[0.61859167979337,-0.623266759536001,0.339563067143743,-0.337016028669028],[0,0,0,0],[8.999999E+09,8.999999E+09,8.999999E+09,8.999999E+09,8.999999E+09,8.999999E+09]];
    LOCAL CONST Robtarget Tr_meulage_motif_1_289 := [[-28.195240234375,-71.3169765625,62.029828125],[0.61859167979337,-0.623266759536001,0.339563067143743,-0.337016028669028],[0,0,0,0],[8.999999E+09,8.999999E+09,8.999999E+09,8.999999E+09,8.999999E+09,8.999999E+09]];
    LOCAL CONST Robtarget Tr_meulage_motif_1_290 := [[-27.644701171875,-72.1517890625,62.029828125],[0.61859167979337,-0.623266759536001,0.339563067143743,-0.337016028669028],[0,0,0,0],[8.999999E+09,8.999999E+09,8.999999E+09,8.999999E+09,8.999999E+09,8.999999E+09]];
    LOCAL CONST Robtarget Tr_meulage_motif_1_291 := [[-27.09416015625,-72.98659375,62.029828125],[0.61859167979337,-0.623266759536001,0.339563067143743,-0.337016028669028],[0,0,0,0],[8.999999E+09,8.999999E+09,8.999999E+09,8.999999E+09,8.999999E+09,8.999999E+09]];
    LOCAL CONST Robtarget Tr_meulage_motif_1_292 := [[-26.54362109375,-73.82140625,62.029828125],[0.61859167979337,-0.623266759536001,0.339563067143743,-0.337016028669028],[0,0,0,0],[8.999999E+09,8.999999E+09,8.999999E+09,8.999999E+09,8.999999E+09,8.999999E+09]];
    LOCAL CONST Robtarget Tr_meulage_motif_1_293 := [[-25.99308203125,-74.6562109375,62.029828125],[0.61859167979337,-0.623266759536001,0.339563067143743,-0.337016028669028],[0,0,0,0],[8.999999E+09,8.999999E+09,8.999999E+09,8.999999E+09,8.999999E+09,8.999999E+09]];
    LOCAL CONST Robtarget Tr_meulage_motif_1_294 := [[-25.442541015625,-75.4910234375,62.029828125],[0.61859167979337,-0.623266759536001,0.339563067143743,-0.337016028669028],[0,0,0,0],[8.999999E+09,8.999999E+09,8.999999E+09,8.999999E+09,8.999999E+09,8.999999E+09]];
    LOCAL CONST Robtarget Tr_meulage_motif_1_295 := [[-24.892001953125,-76.325828125,62.029828125],[0.61859167979337,-0.623266759536001,0.339563067143743,-0.337016028669028],[0,0,0,0],[8.999999E+09,8.999999E+09,8.999999E+09,8.999999E+09,8.999999E+09,8.999999E+09]];
    LOCAL CONST Robtarget Tr_meulage_motif_1_296 := [[-24.3414609375,-77.160640625,62.029828125],[0.61859167979337,-0.623266759536001,0.339563067143743,-0.337016028669028],[0,0,0,0],[8.999999E+09,8.999999E+09,8.999999E+09,8.999999E+09,8.999999E+09,8.999999E+09]];
    LOCAL CONST Robtarget Tr_meulage_motif_1_297 := [[-23.790921875,-77.9954453125,62.029828125],[0.61859167979337,-0.623266759536001,0.339563067143743,-0.337016028669028],[0,0,0,0],[8.999999E+09,8.999999E+09,8.999999E+09,8.999999E+09,8.999999E+09,8.999999E+09]];
    LOCAL CONST Robtarget Tr_meulage_motif_1_298 := [[-23.2403828125,-78.8302578125,62.029828125],[0.61859167979337,-0.623266759536001,0.339563067143743,-0.337016028669028],[0,0,0,0],[8.999999E+09,8.999999E+09,8.999999E+09,8.999999E+09,8.999999E+09,8.999999E+09]];
    LOCAL CONST Robtarget Tr_meulage_motif_1_299 := [[-22.689841796875,-79.6650625,62.029828125],[0.61859167979337,-0.623266759536001,0.339563067143743,-0.337016028669028],[0,0,0,0],[8.999999E+09,8.999999E+09,8.999999E+09,8.999999E+09,8.999999E+09,8.999999E+09]];
    LOCAL CONST Robtarget Tr_meulage_motif_1_300 := [[-22.139302734375,-80.499875,62.029828125],[0.61859167979337,-0.623266759536001,0.339563067143743,-0.337016028669028],[0,0,0,0],[8.999999E+09,8.999999E+09,8.999999E+09,8.999999E+09,8.999999E+09,8.999999E+09]];
    LOCAL CONST Robtarget Tr_meulage_motif_1_301 := [[-21.58876171875,-81.3346796875,62.029828125],[0.61859167979337,-0.623266759536001,0.339563067143743,-0.337016028669028],[0,0,0,0],[8.999999E+09,8.999999E+09,8.999999E+09,8.999999E+09,8.999999E+09,8.999999E+09]];
    LOCAL CONST Robtarget Tr_meulage_motif_1_302 := [[-21.03822265625,-82.1694921875,62.029828125],[0.61859167979337,-0.623266759536001,0.339563067143743,-0.337016028669028],[0,0,0,0],[8.999999E+09,8.999999E+09,8.999999E+09,8.999999E+09,8.999999E+09,8.999999E+09]];
    LOCAL CONST Robtarget Tr_meulage_motif_1_303 := [[-20.48768359375,-83.0043046875,62.029828125],[0.61859167979337,-0.623266759536001,0.339563067143743,-0.337016028669028],[0,0,0,0],[8.999999E+09,8.999999E+09,8.999999E+09,8.999999E+09,8.999999E+09,8.999999E+09]];
    LOCAL CONST Robtarget Tr_meulage_motif_1_304 := [[-19.937142578125,-83.839109375,62.029828125],[0.61859167979337,-0.623266759536001,0.339563067143743,-0.337016028669028],[0,0,0,0],[8.999999E+09,8.999999E+09,8.999999E+09,8.999999E+09,8.999999E+09,8.999999E+09]];
    LOCAL CONST Robtarget Tr_meulage_motif_1_305 := [[-19.386603515625,-84.673921875,62.029828125],[0.61859167979337,-0.623266759536001,0.339563067143743,-0.337016028669028],[0,0,0,0],[8.999999E+09,8.999999E+09,8.999999E+09,8.999999E+09,8.999999E+09,8.999999E+09]];
    LOCAL CONST Robtarget Tr_meulage_motif_1_306 := [[-18.8360625,-85.5087265625,62.029828125],[0.61859167979337,-0.623266759536001,0.339563067143743,-0.337016028669028],[0,0,0,0],[8.999999E+09,8.999999E+09,8.999999E+09,8.999999E+09,8.999999E+09,8.999999E+09]];
    LOCAL CONST Robtarget Tr_meulage_motif_1_307 := [[-18.2855234375,-86.3435390625,62.029828125],[0.61859167979337,-0.623266759536001,0.339563067143743,-0.337016028669028],[0,0,0,0],[8.999999E+09,8.999999E+09,8.999999E+09,8.999999E+09,8.999999E+09,8.999999E+09]];
    LOCAL CONST Robtarget Tr_meulage_motif_1_308 := [[-17.734982421875,-87.17834375,62.029828125],[0.61859167979337,-0.623266759536001,0.339563067143743,-0.337016028669028],[0,0,0,0],[8.999999E+09,8.999999E+09,8.999999E+09,8.999999E+09,8.999999E+09,8.999999E+09]];
    LOCAL CONST Robtarget Tr_meulage_motif_1_309 := [[-17.184443359375,-88.01315625,62.02983203125],[0.61859167979337,-0.623266759536001,0.339563067143743,-0.337016028669028],[0,0,0,0],[8.999999E+09,8.999999E+09,8.999999E+09,8.999999E+09,8.999999E+09,8.999999E+09]];
    LOCAL CONST Robtarget Tr_meulage_motif_1_310 := [[-16.633904296875,-88.8479609375,62.02983203125],[0.61859167979337,-0.623266759536001,0.339563067143743,-0.337016028669028],[0,0,0,0],[8.999999E+09,8.999999E+09,8.999999E+09,8.999999E+09,8.999999E+09,8.999999E+09]];
    LOCAL CONST Robtarget Tr_meulage_motif_1_311 := [[-16.08336328125,-89.6827734375,62.02983203125],[0.61859167979337,-0.623266759536001,0.339563067143743,-0.337016028669028],[0,0,0,0],[8.999999E+09,8.999999E+09,8.999999E+09,8.999999E+09,8.999999E+09,8.999999E+09]];
    LOCAL CONST Robtarget Tr_meulage_motif_1_312 := [[-15.53282421875,-90.517578125,62.02983203125],[0.61859167979337,-0.623266759536001,0.339563067143743,-0.337016028669028],[0,0,0,0],[8.999999E+09,8.999999E+09,8.999999E+09,8.999999E+09,8.999999E+09,8.999999E+09]];
    LOCAL CONST Robtarget Tr_meulage_motif_1_313 := [[-14.9822841796875,-91.352390625,62.02983203125],[0.61859167979337,-0.623266759536001,0.339563067143743,-0.337016028669028],[0,0,0,0],[8.999999E+09,8.999999E+09,8.999999E+09,8.999999E+09,8.999999E+09,8.999999E+09]];
    LOCAL CONST Robtarget Tr_meulage_motif_1_314 := [[-14.431744140625,-92.1871953125,62.02983203125],[0.61859167979337,-0.623266759536001,0.339563067143743,-0.337016028669028],[0,0,0,0],[8.999999E+09,8.999999E+09,8.999999E+09,8.999999E+09,8.999999E+09,8.999999E+09]];
    LOCAL CONST Robtarget Tr_meulage_motif_1_315 := [[-13.8812041015625,-93.0220078125,62.02983203125],[0.61859167979337,-0.623266759536001,0.339563067143743,-0.337016028669028],[0,0,0,0],[8.999999E+09,8.999999E+09,8.999999E+09,8.999999E+09,8.999999E+09,8.999999E+09]];
    LOCAL CONST Robtarget Tr_meulage_motif_1_316 := [[-13.3306640625,-93.8568203125,62.02983203125],[0.61859167979337,-0.623266759536001,0.339563067143743,-0.337016028669028],[0,0,0,0],[8.999999E+09,8.999999E+09,8.999999E+09,8.999999E+09,8.999999E+09,8.999999E+09]];
    LOCAL CONST Robtarget Tr_meulage_motif_1_317 := [[-12.780125,-94.691625,62.02983203125],[0.61859167979337,-0.623266759536001,0.339563067143743,-0.337016028669028],[0,0,0,0],[8.999999E+09,8.999999E+09,8.999999E+09,8.999999E+09,8.999999E+09,8.999999E+09]];
    LOCAL CONST Robtarget Tr_meulage_motif_1_318 := [[-12.2295849609375,-95.5264375,62.02983203125],[0.61859167979337,-0.623266759536001,0.339563067143743,-0.337016028669028],[0,0,0,0],[8.999999E+09,8.999999E+09,8.999999E+09,8.999999E+09,8.999999E+09,8.999999E+09]];
    LOCAL CONST Robtarget Tr_meulage_motif_1_319 := [[-11.679044921875,-96.3612421875,62.02983203125],[0.61859167979337,-0.623266759536001,0.339563067143743,-0.337016028669028],[0,0,0,0],[8.999999E+09,8.999999E+09,8.999999E+09,8.999999E+09,8.999999E+09,8.999999E+09]];
    LOCAL CONST Robtarget Tr_meulage_motif_1_320 := [[-11.1285048828125,-97.1960546875,62.02983203125],[0.61859167979337,-0.623266759536001,0.339563067143743,-0.337016028669028],[0,0,0,0],[8.999999E+09,8.999999E+09,8.999999E+09,8.999999E+09,8.999999E+09,8.999999E+09]];
    LOCAL CONST Robtarget Tr_meulage_motif_1_321 := [[-10.57796484375,-98.030859375,62.02983203125],[0.61859167979337,-0.623266759536001,0.339563067143743,-0.337016028669028],[0,0,0,0],[8.999999E+09,8.999999E+09,8.999999E+09,8.999999E+09,8.999999E+09,8.999999E+09]];
    LOCAL CONST Robtarget Tr_meulage_motif_1_322 := [[-10.03163671875,-98.8595390625,61.91922265625],[0.61859167979337,-0.623266759536001,0.339563067143743,-0.337016028669028],[0,0,0,0],[8.999999E+09,8.999999E+09,8.999999E+09,8.999999E+09,8.999999E+09,8.999999E+09]];
    LOCAL CONST Robtarget Tr_meulage_motif_1_323 := [[-9.5107744140625,-99.6498359375,61.70803515625],[0.61859167979337,-0.623266759536001,0.339563067143743,-0.337016028669028],[0,0,0,0],[8.999999E+09,8.999999E+09,8.999999E+09,8.999999E+09,8.999999E+09,8.999999E+09]];
    LOCAL CONST Robtarget Tr_meulage_motif_1_324 := [[-9.041607421875,-100.3618828125,61.43620703125],[0.61859167979337,-0.623266759536001,0.339563067143743,-0.337016028669028],[0,0,0,0],[8.999999E+09,8.999999E+09,8.999999E+09,8.999999E+09,8.999999E+09,8.999999E+09]];
    LOCAL CONST Robtarget Tr_meulage_motif_1_325 := [[-8.629029296875,-100.988125,61.16026953125],[0.61859167979337,-0.623266759536001,0.339563067143743,-0.337016028669028],[0,0,0,0],[8.999999E+09,8.999999E+09,8.999999E+09,8.999999E+09,8.999999E+09,8.999999E+09]];
    LOCAL CONST Robtarget Tr_meulage_motif_1_326 := [[-8.02350244140625,-101.907734375,60.54414453125],[0.61859167979337,-0.623266759536001,0.339563067143743,-0.337016028669028],[0,0,0,0],[8.999999E+09,8.999999E+09,8.999999E+09,8.999999E+09,8.999999E+09,8.999999E+09]];
    LOCAL CONST Robtarget Tr_meulage_motif_1_327 := [[-7.460716796875,-102.7630625,59.6965078125],[0.61859167979337,-0.623266759536001,0.339563067143743,-0.337016028669028],[0,0,0,0],[8.999999E+09,8.999999E+09,8.999999E+09,8.999999E+09,8.999999E+09,8.999999E+09]];
    LOCAL CONST Robtarget Tr_meulage_motif_1_328 := [[-6.9951328125,-103.4714140625,58.6726484375],[0.61859167979337,-0.623266759536001,0.339563067143743,-0.337016028669028],[0,0,0,0],[8.999999E+09,8.999999E+09,8.999999E+09,8.999999E+09,8.999999E+09,8.999999E+09]];
    LOCAL CONST Robtarget Tr_meulage_motif_1_329 := [[-6.7275654296875,-103.8797109375,57.5564140625],[0.61859167979337,-0.623266759536001,0.339563067143743,-0.337016028669028],[0,0,0,0],[8.999999E+09,8.999999E+09,8.999999E+09,8.999999E+09,8.999999E+09,8.999999E+09]];
    LOCAL CONST Robtarget Tr_meulage_motif_1_330 := [[-6.71340380859375,-103.9027890625,56.8604765625],[0.61859167979337,-0.623266759536001,0.339563067143743,-0.337016028669028],[0,0,0,0],[8.999999E+09,8.999999E+09,8.999999E+09,8.999999E+09,8.999999E+09,8.999999E+09]];
    LOCAL CONST Robtarget Tr_meulage_motif_1_331 := [[-6.7141044921875,-103.90325,56.1991953125],[0.61859167979337,-0.623266759536001,0.339563067143743,-0.337016028669028],[0,0,0,0],[8.999999E+09,8.999999E+09,8.999999E+09,8.999999E+09,8.999999E+09,8.999999E+09]];
    LOCAL CONST Robtarget Tr_meulage_motif_1_332 := [[-6.745015625,-103.8578984375,55.5381171875],[0.61859167979337,-0.623266759536001,0.339563067143743,-0.337016028669028],[0,0,0,0],[8.999999E+09,8.999999E+09,8.999999E+09,8.999999E+09,8.999999E+09,8.999999E+09]];
    LOCAL CONST Robtarget Tr_meulage_motif_1_333 := [[-7.0204716796875,-103.4427578125,54.43638671875],[0.61859167979337,-0.623266759536001,0.339563067143743,-0.337016028669028],[0,0,0,0],[8.999999E+09,8.999999E+09,8.999999E+09,8.999999E+09,8.999999E+09,8.999999E+09]];
    LOCAL CONST Robtarget Tr_meulage_motif_1_334 := [[-7.49314453125,-102.7283359375,53.42974609375],[0.61859167979337,-0.623266759536001,0.339563067143743,-0.337016028669028],[0,0,0,0],[8.999999E+09,8.999999E+09,8.999999E+09,8.999999E+09,8.999999E+09,8.999999E+09]];
    LOCAL CONST Robtarget Tr_meulage_motif_1_335 := [[-8.05746533203125,-101.874546875,52.60088671875],[0.61859167979337,-0.623266759536001,0.339563067143743,-0.337016028669028],[0,0,0,0],[8.999999E+09,8.999999E+09,8.999999E+09,8.999999E+09,8.999999E+09,8.999999E+09]];
    LOCAL CONST Robtarget Tr_meulage_motif_1_336 := [[-8.4361396484375,-101.3012578125,52.20512109375],[0.61859167979337,-0.623266759536001,0.339563067143743,-0.337016028669028],[0,0,0,0],[8.999999E+09,8.999999E+09,8.999999E+09,8.999999E+09,8.999999E+09,8.999999E+09]];
    LOCAL CONST Robtarget Tr_meulage_motif_1_337 := [[-9.074267578125,-100.3347578125,51.71758984375],[0.61859167979337,-0.623266759536001,0.339563067143743,-0.337016028669028],[0,0,0,0],[8.999999E+09,8.999999E+09,8.999999E+09,8.999999E+09,8.999999E+09,8.999999E+09]];
    LOCAL CONST Robtarget Tr_meulage_motif_1_338 := [[-9.5397705078125,-99.6295,51.45348046875],[0.61859167979337,-0.623266759536001,0.339563067143743,-0.337016028669028],[0,0,0,0],[8.999999E+09,8.999999E+09,8.999999E+09,8.999999E+09,8.999999E+09,8.999999E+09]];
    LOCAL CONST Robtarget Tr_meulage_motif_1_339 := [[-10.0530908203125,-98.8516015625,51.24899609375],[0.61859167979337,-0.623266759536001,0.339563067143743,-0.337016028669028],[0,0,0,0],[8.999999E+09,8.999999E+09,8.999999E+09,8.999999E+09,8.999999E+09,8.999999E+09]];
    LOCAL CONST Robtarget Tr_meulage_motif_1_340 := [[-10.5935947265625,-98.0322578125,51.14044921875],[0.61859167979337,-0.623266759536001,0.339563067143743,-0.337016028669028],[0,0,0,0],[8.999999E+09,8.999999E+09,8.999999E+09,8.999999E+09,8.999999E+09,8.999999E+09]];
    LOCAL CONST Robtarget Tr_meulage_motif_1_341 := [[-11.1401572265625,-97.203734375,51.02983984375],[0.61859167979337,-0.623266759536001,0.339563067143743,-0.337016028669028],[0,0,0,0],[8.999999E+09,8.999999E+09,8.999999E+09,8.999999E+09,8.999999E+09,8.999999E+09]];
    LOCAL CONST Robtarget Tr_meulage_motif_1_342 := [[-11.690697265625,-96.3689296875,51.02983984375],[0.61859167979337,-0.623266759536001,0.339563067143743,-0.337016028669028],[0,0,0,0],[8.999999E+09,8.999999E+09,8.999999E+09,8.999999E+09,8.999999E+09,8.999999E+09]];
    LOCAL CONST Robtarget Tr_meulage_motif_1_343 := [[-12.2412373046875,-95.5341171875,51.02983984375],[0.61859167979337,-0.623266759536001,0.339563067143743,-0.337016028669028],[0,0,0,0],[8.999999E+09,8.999999E+09,8.999999E+09,8.999999E+09,8.999999E+09,8.999999E+09]];
    LOCAL CONST Robtarget Tr_meulage_motif_1_344 := [[-12.7917763671875,-94.6993125,51.02983984375],[0.61859167979337,-0.623266759536001,0.339563067143743,-0.337016028669028],[0,0,0,0],[8.999999E+09,8.999999E+09,8.999999E+09,8.999999E+09,8.999999E+09,8.999999E+09]];
    LOCAL CONST Robtarget Tr_meulage_motif_1_345 := [[-13.34231640625,-93.8645,51.02983984375],[0.61859167979337,-0.623266759536001,0.339563067143743,-0.337016028669028],[0,0,0,0],[8.999999E+09,8.999999E+09,8.999999E+09,8.999999E+09,8.999999E+09,8.999999E+09]];
    LOCAL CONST Robtarget Tr_meulage_motif_1_346 := [[-13.8928564453125,-93.0296953125,51.02983984375],[0.61859167979337,-0.623266759536001,0.339563067143743,-0.337016028669028],[0,0,0,0],[8.999999E+09,8.999999E+09,8.999999E+09,8.999999E+09,8.999999E+09,8.999999E+09]];
    LOCAL CONST Robtarget Tr_meulage_motif_1_347 := [[-14.443396484375,-92.1948828125,51.02983984375],[0.61859167979337,-0.623266759536001,0.339563067143743,-0.337016028669028],[0,0,0,0],[8.999999E+09,8.999999E+09,8.999999E+09,8.999999E+09,8.999999E+09,8.999999E+09]];
    LOCAL CONST Robtarget Tr_meulage_motif_1_348 := [[-14.9939365234375,-91.360078125,51.02983984375],[0.61859167979337,-0.623266759536001,0.339563067143743,-0.337016028669028],[0,0,0,0],[8.999999E+09,8.999999E+09,8.999999E+09,8.999999E+09,8.999999E+09,8.999999E+09]];
    LOCAL CONST Robtarget Tr_meulage_motif_1_349 := [[-15.5444765625,-90.525265625,51.02983984375],[0.61859167979337,-0.623266759536001,0.339563067143743,-0.337016028669028],[0,0,0,0],[8.999999E+09,8.999999E+09,8.999999E+09,8.999999E+09,8.999999E+09,8.999999E+09]];
    LOCAL CONST Robtarget Tr_meulage_motif_1_350 := [[-16.095015625,-89.6904609375,51.02983984375],[0.61859167979337,-0.623266759536001,0.339563067143743,-0.337016028669028],[0,0,0,0],[8.999999E+09,8.999999E+09,8.999999E+09,8.999999E+09,8.999999E+09,8.999999E+09]];
    LOCAL CONST Robtarget Tr_meulage_motif_1_351 := [[-16.645556640625,-88.8556484375,51.02983984375],[0.61859167979337,-0.623266759536001,0.339563067143743,-0.337016028669028],[0,0,0,0],[8.999999E+09,8.999999E+09,8.999999E+09,8.999999E+09,8.999999E+09,8.999999E+09]];
    LOCAL CONST Robtarget Tr_meulage_motif_1_352 := [[-17.196095703125,-88.02084375,51.02983984375],[0.61859167979337,-0.623266759536001,0.339563067143743,-0.337016028669028],[0,0,0,0],[8.999999E+09,8.999999E+09,8.999999E+09,8.999999E+09,8.999999E+09,8.999999E+09]];
    LOCAL CONST Robtarget Tr_meulage_motif_1_353 := [[-17.746634765625,-87.18603125,51.02983984375],[0.61859167979337,-0.623266759536001,0.339563067143743,-0.337016028669028],[0,0,0,0],[8.999999E+09,8.999999E+09,8.999999E+09,8.999999E+09,8.999999E+09,8.999999E+09]];
    LOCAL CONST Robtarget Tr_meulage_motif_1_354 := [[-18.29717578125,-86.35121875,51.02983984375],[0.61859167979337,-0.623266759536001,0.339563067143743,-0.337016028669028],[0,0,0,0],[8.999999E+09,8.999999E+09,8.999999E+09,8.999999E+09,8.999999E+09,8.999999E+09]];
    LOCAL CONST Robtarget Tr_meulage_motif_1_355 := [[-18.84771484375,-85.5164140625,51.02983984375],[0.61859167979337,-0.623266759536001,0.339563067143743,-0.337016028669028],[0,0,0,0],[8.999999E+09,8.999999E+09,8.999999E+09,8.999999E+09,8.999999E+09,8.999999E+09]];
    LOCAL CONST Robtarget Tr_meulage_motif_1_356 := [[-19.398255859375,-84.6816015625,51.02983984375],[0.61859167979337,-0.623266759536001,0.339563067143743,-0.337016028669028],[0,0,0,0],[8.999999E+09,8.999999E+09,8.999999E+09,8.999999E+09,8.999999E+09,8.999999E+09]];
    LOCAL CONST Robtarget Tr_meulage_motif_1_357 := [[-19.948794921875,-83.846796875,51.02983984375],[0.61859167979337,-0.623266759536001,0.339563067143743,-0.337016028669028],[0,0,0,0],[8.999999E+09,8.999999E+09,8.999999E+09,8.999999E+09,8.999999E+09,8.999999E+09]];
    LOCAL CONST Robtarget Tr_meulage_motif_1_358 := [[-20.4993359375,-83.011984375,51.02983984375],[0.61859167979337,-0.623266759536001,0.339563067143743,-0.337016028669028],[0,0,0,0],[8.999999E+09,8.999999E+09,8.999999E+09,8.999999E+09,8.999999E+09,8.999999E+09]];
    LOCAL CONST Robtarget Tr_meulage_motif_1_359 := [[-21.049875,-82.1771796875,51.02983984375],[0.61859167979337,-0.623266759536001,0.339563067143743,-0.337016028669028],[0,0,0,0],[8.999999E+09,8.999999E+09,8.999999E+09,8.999999E+09,8.999999E+09,8.999999E+09]];
    LOCAL CONST Robtarget Tr_meulage_motif_1_360 := [[-21.6004140625,-81.3423671875,51.02983984375],[0.61859167979337,-0.623266759536001,0.339563067143743,-0.337016028669028],[0,0,0,0],[8.999999E+09,8.999999E+09,8.999999E+09,8.999999E+09,8.999999E+09,8.999999E+09]];
    LOCAL CONST Robtarget Tr_meulage_motif_1_361 := [[-22.150955078125,-80.5075625,51.02983984375],[0.61859167979337,-0.623266759536001,0.339563067143743,-0.337016028669028],[0,0,0,0],[8.999999E+09,8.999999E+09,8.999999E+09,8.999999E+09,8.999999E+09,8.999999E+09]];
    LOCAL CONST Robtarget Tr_meulage_motif_1_362 := [[-22.701494140625,-79.67275,51.0298359375],[0.61859167979337,-0.623266759536001,0.339563067143743,-0.337016028669028],[0,0,0,0],[8.999999E+09,8.999999E+09,8.999999E+09,8.999999E+09,8.999999E+09,8.999999E+09]];
    LOCAL CONST Robtarget Tr_meulage_motif_1_363 := [[-23.25203515625,-78.8379453125,51.0298359375],[0.61859167979337,-0.623266759536001,0.339563067143743,-0.337016028669028],[0,0,0,0],[8.999999E+09,8.999999E+09,8.999999E+09,8.999999E+09,8.999999E+09,8.999999E+09]];
    LOCAL CONST Robtarget Tr_meulage_motif_1_364 := [[-23.80257421875,-78.0031328125,51.0298359375],[0.61859167979337,-0.623266759536001,0.339563067143743,-0.337016028669028],[0,0,0,0],[8.999999E+09,8.999999E+09,8.999999E+09,8.999999E+09,8.999999E+09,8.999999E+09]];
    LOCAL CONST Robtarget Tr_meulage_motif_1_365 := [[-24.35311328125,-77.168328125,51.0298359375],[0.61859167979337,-0.623266759536001,0.339563067143743,-0.337016028669028],[0,0,0,0],[8.999999E+09,8.999999E+09,8.999999E+09,8.999999E+09,8.999999E+09,8.999999E+09]];
    LOCAL CONST Robtarget Tr_meulage_motif_1_366 := [[-24.903654296875,-76.333515625,51.0298359375],[0.61859167979337,-0.623266759536001,0.339563067143743,-0.337016028669028],[0,0,0,0],[8.999999E+09,8.999999E+09,8.999999E+09,8.999999E+09,8.999999E+09,8.999999E+09]];
    LOCAL CONST Robtarget Tr_meulage_motif_1_367 := [[-25.454193359375,-75.4987109375,51.0298359375],[0.61859167979337,-0.623266759536001,0.339563067143743,-0.337016028669028],[0,0,0,0],[8.999999E+09,8.999999E+09,8.999999E+09,8.999999E+09,8.999999E+09,8.999999E+09]];
    LOCAL CONST Robtarget Tr_meulage_motif_1_368 := [[-26.004734375,-74.6638984375,51.0298359375],[0.61859167979337,-0.623266759536001,0.339563067143743,-0.337016028669028],[0,0,0,0],[8.999999E+09,8.999999E+09,8.999999E+09,8.999999E+09,8.999999E+09,8.999999E+09]];
    LOCAL CONST Robtarget Tr_meulage_motif_1_369 := [[-26.5552734375,-73.8290859375,51.0298359375],[0.61859167979337,-0.623266759536001,0.339563067143743,-0.337016028669028],[0,0,0,0],[8.999999E+09,8.999999E+09,8.999999E+09,8.999999E+09,8.999999E+09,8.999999E+09]];
    LOCAL CONST Robtarget Tr_meulage_motif_1_370 := [[-27.1058125,-72.99428125,51.0298359375],[0.61859167979337,-0.623266759536001,0.339563067143743,-0.337016028669028],[0,0,0,0],[8.999999E+09,8.999999E+09,8.999999E+09,8.999999E+09,8.999999E+09,8.999999E+09]];
    LOCAL CONST Robtarget Tr_meulage_motif_1_371 := [[-27.656353515625,-72.15946875,51.0298359375],[0.61859167979337,-0.623266759536001,0.339563067143743,-0.337016028669028],[0,0,0,0],[8.999999E+09,8.999999E+09,8.999999E+09,8.999999E+09,8.999999E+09,8.999999E+09]];
